KUKA KRL program: EPS_2_25694_RR02_A_20260114065911.src

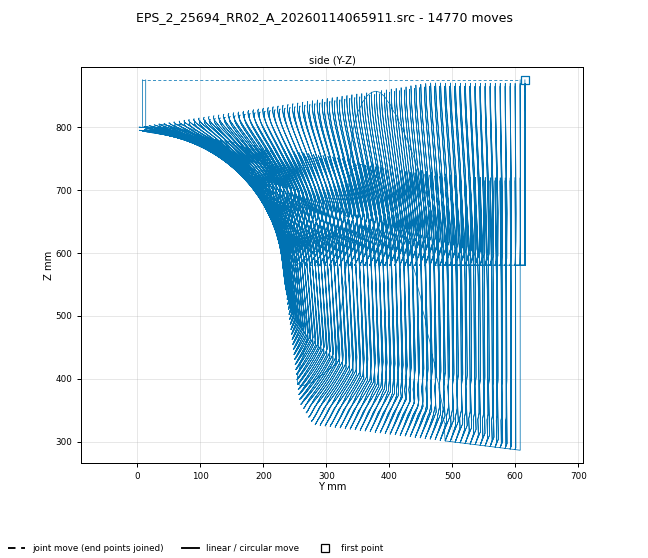
[picture p0: tool path of EPS_2_25694_RR02_A_20260114065911.src, 14770 of 14772 moves have a stored position in this frame; points joined in program order, loops and branches not executed]
&ACCESS RVP
&REL 4
&COMMENT QRS 19112012
&PARAM EDITMASK = *
DEF PART()
EXT BAS (BAS_COMMAND :IN,REAL :IN )
INT I
BAS (#INITMOV,0 )

;KUKA QRS Post kuka4.cps  Date:22-06-2017 !

File_ID=2963

QRS_PRE_INIT()

;Init var - Until changes are made in qrs_pre_init
Outlet_Square_prg=0
Inlet_1_Square_prg=0
Inlet_2_Square_prg=0
Inlet_3_Square_prg=0
Inlet_4_Square_prg=0
Inlet_5_Square_prg=0

Outlet_1={X 0.000, Y 466.000, Z 636.500, B 0.000, E1 0.000 }
Inlet_1={X 0.000, Y 521.440, Z 392.000, B 0.000, E1 180.000 }
Outlet_1_type=457
Inlet_1_type=366
;QRS#1=Sidecore dimensions
;QRS#2=450-18" Concrete
;QRS#3=375-15" PVC SDR 35
;QRS#4=
;QRS#5=
;QRS#6=
;QRS#7=
;QRS#8=
;QRS#9=28A PSX-2
;QRS#10=20Y PSX
;QRS#11=
;QRS#12=
;QRS#13=
;QRS#14=
;QRS#15=
;QRS#16=1220x127x1219 4'
;QRS#17=EPS Height
;QRS#18=865
;QRS#19=*
;QRS#20= UPDATED VERSION 22-06-2017
;QRS#21=*
Outlet_Square=0250
Inlet_1_Square=0250
Inlet_2_Square=0
Inlet_3_Square=0
Inlet_4_Square=0
Inlet_5_Square=0
Mill_Square=1
Outlet_Square_Prg=274
Inlet_1_Square_prg=252

QRS_INIT()

$ADVANCE=5

; T1
PTP {E1 172.637,E2 172.637}
PTP {X 0,Y 615.384,A -85,B 0,C 180,E1 172.637,E2 172.637,E3 0,E4 0,E5 0,E6 0}
QRS_SPEED_INIT()
LIN {X 0,Y 615.384,Z 875,A -85,B 0,C 180,E1 172.637,E2 172.637,E3 0,E4 0,E5 0,E6 0} C_VEL
LIN {X 0,Y 615.384,Z 582.66,A -85,B 0,C 180,E1 172.637,E2 172.637} C_VEL
LIN {X 0,Y 615.412,Z 580.66,A -85,B 0,C 180,E1 172.823,E2 172.823} C_VEL
LIN {X 0,Y 615.825,Z 580.66,A -85,B 0,C 180,E1 174.193,E2 174.193} C_VEL
LIN {X 0,Y 615.841,Z 580.66,A -85,B 0,C 180,E1 178.841,E2 178.841} C_VEL
LIN {X 0,Y 615.793,Z 580.66,A -85,B 0,C 180,E1 183.481,E2 183.481} C_VEL
LIN {X 0,Y 615.82,Z 580.66,A -85,B 0,C 180,E1 188.143,E2 188.143} C_VEL
LIN {X 0,Y 615.802,Z 580.66,A -85,B 0,C 180,E1 192.862,E2 192.862} C_VEL
LIN {X 0,Y 615.751,Z 580.66,A -85,B 0,C 180,E1 197.672,E2 197.672} C_VEL
LIN {X 0,Y 615.756,Z 580.66,A -85,B 0,C 180,E1 197.985,E2 197.985} C_VEL
LIN {X 0,Y 615.766,Z 580.66,A -85,B 0,C 180,E1 202.613,E2 202.613} C_VEL
LIN {X 0,Y 615.233,Z 580.66,A -85,B 0,C 180,E1 205.173,E2 205.173} C_VEL
LIN {X 0,Y 615.723,Z 580.66,A -85,B 0,C 180,E1 207.742,E2 207.742} C_VEL
LIN {X 0,Y 615.16,Z 580.66,A -85,B 0,C 180,E1 210.426,E2 210.426} C_VEL
LIN {X 0,Y 615.691,Z 580.66,A -85,B 0,C 180,E1 213.125,E2 213.125} C_VEL
LIN {X 0,Y 615.621,Z 580.66,A -85,B 0,C 180,E1 213.912,E2 213.912} C_VEL
LIN {X 0,Y 615.656,Z 580.66,A -85,B 0,C 180,E1 218.863,E2 218.863} C_VEL
LIN {X 0,Y 615.25,Z 580.66,A -85,B 0,C 180,E1 221.943,E2 221.943} C_VEL
LIN {X 0,Y 615.658,Z 580.66,A -85,B 0,C 180,E1 224.895,E2 224.895} C_VEL
LIN {X 0,Y 615.649,Z 580.66,A -85,B 0,C 180,E1 228.497,E2 228.497} C_VEL
LIN {X 0,Y 615.377,Z 580.66,A -85,B 0,C 180,E1 231.117,E2 231.117} C_VEL
LIN {X 0,Y 615.425,Z 580.66,A -85,B 0,C 180,E1 232.156,E2 232.156} C_VEL
LIN {X 0,Y 615.687,Z 580.66,A -85,B 0,C 180,E1 234.06,E2 234.06} C_VEL
LIN {X 0,Y 615.153,Z 580.66,A -85,B 0,C 180,E1 236.843,E2 236.843} C_VEL
LIN {X 0,Y 615.758,Z 580.66,A -85,B 0,C 180,E1 239.607,E2 239.607} C_VEL
LIN {X 0,Y 615.721,Z 580.66,A -85,B 0,C 180,E1 243.936,E2 243.936} C_VEL
LIN {X 0,Y 615.733,Z 580.66,A -85,B 0,C 180,E1 244.38,E2 244.38} C_VEL
LIN {X 0,Y 614.989,Z 580.66,A -85,B 0,C 180,E1 244.523,E2 244.523} C_VEL
LIN {X 0,Y 614.799,Z 580.769,A -85,B 0,C 180,E1 244.548,E2 244.548} C_VEL
LIN {X 0,Y 615.5,Z 597.034,A -85,B 0,C 180,E1 244.785,E2 244.785} C_VEL
LIN {X 0,Y 615.746,Z 643.934,A -85,B 0,C 180,E1 245.388,E2 245.388} C_VEL
LIN {X 0,Y 615.746,Z 656.529,A -85,B 0,C 180,E1 245.585,E2 245.585} C_VEL
LIN {X 0,Y 615.551,Z 668.878,A -85,B 0,C 180,E1 245.832,E2 245.832} C_VEL
LIN {X 0,Y 615.688,Z 680.202,A -85,B 0,C 180,E1 246.128,E2 246.128} C_VEL
LIN {X 0,Y 615.662,Z 691.181,A -85,B 0,C 180,E1 246.461,E2 246.461} C_VEL
LIN {X 0,Y 615.686,Z 701.114,A -85,B 0,C 180,E1 246.809,E2 246.809} C_VEL
LIN {X 0,Y 615.746,Z 713.854,A -85,B 0,C 180,E1 247.329,E2 247.329} C_VEL
LIN {X 0,Y 615.681,Z 724.625,A -85,B 0,C 180,E1 247.824,E2 247.824} C_VEL
LIN {X 0,Y 615.745,Z 734.343,A -85,B 0,C 180,E1 248.326,E2 248.326} C_VEL
LIN {X 0,Y 615.763,Z 745.218,A -85,B 0,C 180,E1 248.949,E2 248.949} C_VEL
LIN {X 0,Y 615.754,Z 755.026,A -85,B 0,C 180,E1 249.568,E2 249.568} C_VEL
LIN {X 0,Y 615.75,Z 764.993,A -85,B 0,C 180,E1 250.263,E2 250.263} C_VEL
LIN {X 0,Y 615.755,Z 774.06,A -85,B 0,C 180,E1 250.954,E2 250.954} C_VEL
LIN {X 0,Y 615.778,Z 783.429,A -85,B 0,C 180,E1 251.737,E2 251.737} C_VEL
LIN {X 0,Y 615.741,Z 791.079,A -85,B 0,C 180,E1 252.429,E2 252.429} C_VEL
LIN {X 0,Y 615.699,Z 798.268,A -85,B 0,C 180,E1 253.129,E2 253.129} C_VEL
LIN {X 0,Y 615.745,Z 806.234,A -85,B 0,C 180,E1 253.979,E2 253.979} C_VEL
LIN {X 0,Y 615.811,Z 812.886,A -85,B 0,C 180,E1 254.748,E2 254.748} C_VEL
LIN {X 0,Y 615.686,Z 820.033,A -85,B 0,C 180,E1 255.645,E2 255.645} C_VEL
LIN {X 0,Y 615.678,Z 826.532,A -85,B 0,C 180,E1 256.541,E2 256.541} C_VEL
LIN {X 0,Y 615.8,Z 832.432,A -85,B 0,C 180,E1 257.436,E2 257.436} C_VEL
LIN {X 0,Y 615.696,Z 837.811,A -85,B 0,C 180,E1 258.323,E2 258.323} C_VEL
LIN {X 0,Y 615.617,Z 844.151,A -85,B 0,C 180,E1 259.503,E2 259.503} C_VEL
LIN {X 0,Y 615.751,Z 848.397,A -85,B 0,C 180,E1 260.389,E2 260.389} C_VEL
LIN {X 0,Y 615.781,Z 852.167,A -85,B 0,C 180,E1 261.27,E2 261.27} C_VEL
LIN {X 0,Y 615.632,Z 857.066,A -85,B 0,C 180,E1 262.574,E2 262.574} C_VEL
LIN {X 0,Y 615.761,Z 860.68,A -85,B 0,C 180,E1 263.748,E2 263.748} C_VEL
LIN {X 0,Y 615.831,Z 861.858,A -85,B 0,C 180,E1 264.193,E2 264.193} C_VEL
LIN {X 0,Y 615.724,Z 863.1,A -85,B 0,C 180,E1 264.658,E2 264.658} C_VEL
LIN {X 0,Y 615.59,Z 865.15,A -85,B 0,C 180,E1 265.588,E2 265.588} C_VEL
LIN {X 0,Y 615.604,Z 866.752,A -85,B 0,C 180,E1 266.518,E2 266.518} C_VEL
LIN {X 0,Y 615.789,Z 867.942,A -85,B 0,C 180,E1 267.448,E2 267.448} C_VEL
LIN {X 0,Y 615.603,Z 869.162,A -85,B 0,C 180,E1 268.84,E2 268.84} C_VEL
LIN {X 0,Y 615.628,Z 869.418,A -85,B 0,C 180,E1 270.232,E2 270.232} C_VEL
LIN {X 0,Y 615.832,Z 869.118,A -85,B 0,C 180,E1 271.159,E2 271.159} C_VEL
LIN {X 0,Y 615.718,Z 868.484,A -85,B 0,C 180,E1 272.087,E2 272.087} C_VEL
LIN {X 0,Y 615.795,Z 866.717,A -85,B 0,C 180,E1 273.48,E2 273.48} C_VEL
LIN {X 0,Y 615.708,Z 865.13,A -85,B 0,C 180,E1 274.411,E2 274.411} C_VEL
LIN {X 0,Y 615.577,Z 863.127,A -85,B 0,C 180,E1 275.343,E2 275.343} C_VEL
LIN {X 0,Y 615.645,Z 860.601,A -85,B 0,C 180,E1 276.29,E2 276.29} C_VEL
LIN {X 0,Y 615.806,Z 856.594,A -85,B 0,C 180,E1 277.559,E2 277.559} C_VEL
LIN {X 0,Y 615.635,Z 852.191,A -85,B 0,C 180,E1 278.731,E2 278.731} C_VEL
LIN {X 0,Y 615.664,Z 848.411,A -85,B 0,C 180,E1 279.612,E2 279.612} C_VEL
LIN {X 0,Y 615.797,Z 842.63,A -85,B 0,C 180,E1 280.788,E2 280.788} C_VEL
LIN {X 0,Y 615.635,Z 837.82,A -85,B 0,C 180,E1 281.678,E2 281.678} C_VEL
LIN {X 0,Y 615.632,Z 832.452,A -85,B 0,C 180,E1 282.567,E2 282.567} C_VEL
LIN {X 0,Y 615.823,Z 824.412,A -85,B 0,C 180,E1 283.754,E2 283.754} C_VEL
LIN {X 0,Y 615.734,Z 817.716,A -85,B 0,C 180,E1 284.653,E2 284.653} C_VEL
LIN {X 0,Y 615.702,Z 810.34,A -85,B 0,C 180,E1 285.554,E2 285.554} C_VEL
LIN {X 0,Y 615.782,Z 803.643,A -85,B 0,C 180,E1 286.305,E2 286.305} C_VEL
LIN {X 0,Y 615.769,Z 795.301,A -85,B 0,C 180,E1 287.164,E2 287.164} C_VEL
LIN {X 0,Y 615.716,Z 786.769,A -85,B 0,C 180,E1 287.969,E2 287.969} C_VEL
LIN {X 0,Y 615.738,Z 778.66,A -85,B 0,C 180,E1 288.672,E2 288.672} C_VEL
LIN {X 0,Y 615.745,Z 770.145,A -85,B 0,C 180,E1 289.353,E2 289.353} C_VEL
LIN {X 0,Y 615.75,Z 760.692,A -85,B 0,C 180,E1 290.045,E2 290.045} C_VEL
LIN {X 0,Y 615.742,Z 751.477,A -85,B 0,C 180,E1 290.664,E2 290.664} C_VEL
LIN {X 0,Y 615.715,Z 741.286,A -85,B 0,C 180,E1 291.286,E2 291.286} C_VEL
LIN {X 0,Y 615.749,Z 731.423,A -85,B 0,C 180,E1 291.83,E2 291.83} C_VEL
LIN {X 0,Y 615.746,Z 720.95,A -85,B 0,C 180,E1 292.351,E2 292.351} C_VEL
LIN {X 0,Y 615.698,Z 709.84,A -85,B 0,C 180,E1 292.845,E2 292.845} C_VEL
LIN {X 0,Y 615.669,Z 699.566,A -85,B 0,C 180,E1 293.249,E2 293.249} C_VEL
LIN {X 0,Y 615.734,Z 686.394,A -85,B 0,C 180,E1 293.687,E2 293.687} C_VEL
LIN {X 0,Y 615.669,Z 674.855,A -85,B 0,C 180,E1 294.016,E2 294.016} C_VEL
LIN {X 0,Y 615.62,Z 666.572,A -85,B 0,C 180,E1 294.221,E2 294.221} C_VEL
LIN {X 0,Y 615.767,Z 652.574,A -85,B 0,C 180,E1 294.483,E2 294.483} C_VEL
LIN {X 0,Y 615.685,Z 635.543,A -85,B 0,C 180,E1 294.722,E2 294.722} C_VEL
LIN {X 0,Y 615.162,Z 597.63,A -85,B 0,C 180,E1 295.223,E2 295.223} C_VEL
LIN {X 0,Y 614.785,Z 580.66,A -85,B 0,C 180,E1 295.457,E2 295.457} C_VEL
LIN {X 0,Y 615.85,Z 580.66,A -85,B 0,C 180,E1 295.73,E2 295.73} C_VEL
LIN {X 0,Y 615.813,Z 580.66,A -85,B 0,C 180,E1 297.736,E2 297.736} C_VEL
LIN {X 0,Y 615.182,Z 580.66,A -85,B 0,C 180,E1 300.424,E2 300.424} C_VEL
LIN {X 0,Y 615.704,Z 580.66,A -85,B 0,C 180,E1 303.123,E2 303.123} C_VEL
LIN {X 0,Y 615.639,Z 580.66,A -85,B 0,C 180,E1 303.912,E2 303.912} C_VEL
LIN {X 0,Y 615.658,Z 580.66,A -85,B 0,C 180,E1 308.862,E2 308.862} C_VEL
LIN {X 0,Y 615.25,Z 580.66,A -85,B 0,C 180,E1 311.941,E2 311.941} C_VEL
LIN {X 0,Y 615.666,Z 580.66,A -85,B 0,C 180,E1 314.894,E2 314.894} C_VEL
LIN {X 0,Y 615.661,Z 580.66,A -85,B 0,C 180,E1 318.493,E2 318.493} C_VEL
LIN {X 0,Y 615.374,Z 580.66,A -85,B 0,C 180,E1 321.115,E2 321.115} C_VEL
LIN {X 0,Y 615.423,Z 580.66,A -85,B 0,C 180,E1 322.154,E2 322.154} C_VEL
LIN {X 0,Y 615.672,Z 580.66,A -85,B 0,C 180,E1 324.058,E2 324.058} C_VEL
LIN {X 0,Y 615.143,Z 580.66,A -85,B 0,C 180,E1 326.841,E2 326.841} C_VEL
LIN {X 0,Y 615.743,Z 580.66,A -85,B 0,C 180,E1 329.606,E2 329.606} C_VEL
LIN {X 0,Y 615.21,Z 580.66,A -85,B 0,C 180,E1 332.233,E2 332.233} C_VEL
LIN {X 0,Y 615.726,Z 580.66,A -85,B 0,C 180,E1 334.849,E2 334.849} C_VEL
LIN {X 0,Y 615.762,Z 580.66,A -85,B 0,C 180,E1 339.877,E2 339.877} C_VEL
LIN {X 0,Y 615.795,Z 580.66,A -85,B 0,C 180,E1 343.784,E2 343.784} C_VEL
LIN {X 0,Y 615.809,Z 580.66,A -85,B 0,C 180,E1 349.507,E2 349.507} C_VEL
LIN {X 0,Y 615.792,Z 580.66,A -85,B 0,C 180,E1 354.193,E2 354.193} C_VEL
LIN {X 0,Y 615.815,Z 580.66,A -85,B 0,C 180,E1 358.841,E2 358.841} C_VEL
LIN {X 0,Y 615.862,Z 580.66,A -85,B 0,C 180,E1 363.48,E2 363.48} C_VEL
LIN {X 0,Y 615.786,Z 580.66,A -85,B 0,C 180,E1 368.144,E2 368.144} C_VEL
LIN {X 0,Y 615.765,Z 580.66,A -85,B 0,C 180,E1 372.862,E2 372.862} C_VEL
LIN {X 0,Y 615.802,Z 580.66,A -85,B 0,C 180,E1 377.67,E2 377.67} C_VEL
LIN {X 0,Y 615.801,Z 580.66,A -85,B 0,C 180,E1 377.999,E2 377.999} C_VEL
LIN {X 0,Y 615.737,Z 580.66,A -85,B 0,C 180,E1 382.614,E2 382.614} C_VEL
LIN {X 0,Y 615.212,Z 580.66,A -85,B 0,C 180,E1 385.174,E2 385.174} C_VEL
LIN {X 0,Y 615.723,Z 580.66,A -85,B 0,C 180,E1 387.742,E2 387.742} C_VEL
LIN {X 0,Y 615.169,Z 580.66,A -85,B 0,C 180,E1 390.426,E2 390.426} C_VEL
LIN {X 0,Y 615.697,Z 580.66,A -85,B 0,C 180,E1 393.125,E2 393.125} C_VEL
LIN {X 0,Y 615.637,Z 580.66,A -85,B 0,C 180,E1 393.915,E2 393.915} C_VEL
LIN {X 0,Y 615.621,Z 580.66,A -85,B 0,C 180,E1 398.866,E2 398.866} C_VEL
LIN {X 0,Y 615.224,Z 580.66,A -85,B 0,C 180,E1 401.945,E2 401.945} C_VEL
LIN {X 0,Y 615.653,Z 580.66,A -85,B 0,C 180,E1 404.895,E2 404.895} C_VEL
LIN {X 0,Y 615.628,Z 580.66,A -85,B 0,C 180,E1 408.499,E2 408.499} C_VEL
LIN {X 0,Y 615.36,Z 580.66,A -85,B 0,C 180,E1 411.116,E2 411.116} C_VEL
LIN {X 0,Y 615.418,Z 580.66,A -85,B 0,C 180,E1 412.157,E2 412.157} C_VEL
LIN {X 0,Y 615.69,Z 580.66,A -85,B 0,C 180,E1 414.061,E2 414.061} C_VEL
LIN {X 0,Y 615.128,Z 580.66,A -85,B 0,C 180,E1 416.842,E2 416.842} C_VEL
LIN {X 0,Y 615.699,Z 580.66,A -85,B 0,C 180,E1 419.605,E2 419.605} C_VEL
LIN {X 0,Y 615.208,Z 580.66,A -85,B 0,C 180,E1 422.234,E2 422.234} C_VEL
LIN {X 0,Y 615.756,Z 580.66,A -85,B 0,C 180,E1 424.851,E2 424.851} C_VEL
LIN {X 0,Y 615.821,Z 580.66,A -85,B 0,C 180,E1 429.88,E2 429.88} C_VEL
LIN {X 0,Y 615.638,Z 580.69,A -85,B 0,C 180,E1 431.013,E2 431.013} C_VEL
LIN {X 0,Y 615.768,Z 591.798,A -85,B 0,C 180,E1 431.458,E2 431.458} C_VEL
LIN {X 0,Y 615.772,Z 600.905,A -85,B 0,C 180,E1 431.871,E2 431.871} C_VEL
LIN {X 0,Y 615.729,Z 609.887,A -85,B 0,C 180,E1 432.328,E2 432.328} C_VEL
LIN {X 0,Y 615.771,Z 617.761,A -85,B 0,C 180,E1 432.774,E2 432.774} C_VEL
LIN {X 0,Y 615.774,Z 624.953,A -85,B 0,C 180,E1 433.218,E2 433.218} C_VEL
LIN {X 0,Y 615.803,Z 633.619,A -85,B 0,C 180,E1 433.81,E2 433.81} C_VEL
LIN {X 0,Y 615.788,Z 641.35,A -85,B 0,C 180,E1 434.39,E2 434.39} C_VEL
LIN {X 0,Y 615.765,Z 649.322,A -85,B 0,C 180,E1 435.048,E2 435.048} C_VEL
LIN {X 0,Y 615.775,Z 655.958,A -85,B 0,C 180,E1 435.647,E2 435.647} C_VEL
LIN {X 0,Y 615.829,Z 663.488,A -85,B 0,C 180,E1 436.395,E2 436.395} C_VEL
LIN {X 0,Y 615.772,Z 668.99,A -85,B 0,C 180,E1 436.99,E2 436.99} C_VEL
LIN {X 0,Y 615.717,Z 675.289,A -85,B 0,C 180,E1 437.731,E2 437.731} C_VEL
LIN {X 0,Y 615.762,Z 681.001,A -85,B 0,C 180,E1 438.473,E2 438.473} C_VEL
LIN {X 0,Y 615.83,Z 686.181,A -85,B 0,C 180,E1 439.213,E2 439.213} C_VEL
LIN {X 0,Y 615.701,Z 691.8,A -85,B 0,C 180,E1 440.094,E2 440.094} C_VEL
LIN {X 0,Y 615.678,Z 695.184,A -85,B 0,C 180,E1 440.682,E2 440.682} C_VEL
LIN {X 0,Y 615.763,Z 699.755,A -85,B 0,C 180,E1 441.564,E2 441.564} C_VEL
LIN {X 0,Y 615.828,Z 702.587,A -85,B 0,C 180,E1 442.164,E2 442.164} C_VEL
LIN {X 0,Y 615.7,Z 705.584,A -85,B 0,C 180,E1 442.857,E2 442.857} C_VEL
LIN {X 0,Y 615.634,Z 708.833,A -85,B 0,C 180,E1 443.718,E2 443.718} C_VEL
LIN {X 0,Y 615.72,Z 711.829,A -85,B 0,C 180,E1 444.658,E2 444.658} C_VEL
LIN {X 0,Y 615.799,Z 714.279,A -85,B 0,C 180,E1 445.59,E2 445.59} C_VEL
LIN {X 0,Y 615.646,Z 716.272,A -85,B 0,C 180,E1 446.519,E2 446.519} C_VEL
LIN {X 0,Y 615.657,Z 717.751,A -85,B 0,C 180,E1 447.448,E2 447.448} C_VEL
LIN {X 0,Y 615.718,Z 718.288,A -85,B 0,C 180,E1 447.913,E2 447.913} C_VEL
LIN {X 0,Y 615.776,Z 719.068,A -85,B 0,C 180,E1 448.841,E2 448.841} C_VEL
LIN {X 0,Y 615.635,Z 719.428,A -85,B 0,C 180,E1 449.768,E2 449.768} C_VEL
LIN {X 0,Y 615.625,Z 719.408,A -85,B 0,C 180,E1 450.232,E2 450.232} C_VEL
LIN {X 0,Y 615.726,Z 719.014,A -85,B 0,C 180,E1 451.16,E2 451.16} C_VEL
LIN {X 0,Y 615.709,Z 717.635,A -85,B 0,C 180,E1 452.552,E2 452.552} C_VEL
LIN {X 0,Y 615.64,Z 716.119,A -85,B 0,C 180,E1 453.481,E2 453.481} C_VEL
LIN {X 0,Y 615.741,Z 714.08,A -85,B 0,C 180,E1 454.411,E2 454.411} C_VEL
LIN {X 0,Y 615.791,Z 711.544,A -85,B 0,C 180,E1 455.341,E2 455.341} C_VEL
LIN {X 0,Y 615.685,Z 708.479,A -85,B 0,C 180,E1 456.284,E2 456.284} C_VEL
LIN {X 0,Y 615.769,Z 703.979,A -85,B 0,C 180,E1 457.424,E2 457.424} C_VEL
LIN {X 0,Y 615.81,Z 700.733,A -85,B 0,C 180,E1 458.143,E2 458.143} C_VEL
LIN {X 0,Y 615.718,Z 697.886,A -85,B 0,C 180,E1 458.731,E2 458.731} C_VEL
LIN {X 0,Y 615.682,Z 693.041,A -85,B 0,C 180,E1 459.612,E2 459.612} C_VEL
LIN {X 0,Y 615.79,Z 687.56,A -85,B 0,C 180,E1 460.494,E2 460.494} C_VEL
LIN {X 0,Y 615.811,Z 682.514,A -85,B 0,C 180,E1 461.231,E2 461.231} C_VEL
LIN {X 0,Y 615.725,Z 676.961,A -85,B 0,C 180,E1 461.972,E2 461.972} C_VEL
LIN {X 0,Y 615.74,Z 670.826,A -85,B 0,C 180,E1 462.714,E2 462.714} C_VEL
LIN {X 0,Y 615.83,Z 664.055,A -85,B 0,C 180,E1 463.456,E2 463.456} C_VEL
LIN {X 0,Y 615.807,Z 658.152,A -85,B 0,C 180,E1 464.053,E2 464.053} C_VEL
LIN {X 0,Y 615.764,Z 651.723,A -85,B 0,C 180,E1 464.653,E2 464.653} C_VEL
LIN {X 0,Y 615.786,Z 644.696,A -85,B 0,C 180,E1 465.252,E2 465.252} C_VEL
LIN {X 0,Y 615.794,Z 636.939,A -85,B 0,C 180,E1 465.857,E2 465.857} C_VEL
LIN {X 0,Y 615.802,Z 629.564,A -85,B 0,C 180,E1 466.384,E2 466.384} C_VEL
LIN {X 0,Y 615.782,Z 622.271,A -85,B 0,C 180,E1 466.862,E2 466.862} C_VEL
LIN {X 0,Y 615.747,Z 613.78,A -85,B 0,C 180,E1 467.368,E2 467.368} C_VEL
LIN {X 0,Y 615.782,Z 604.229,A -85,B 0,C 180,E1 467.875,E2 467.875} C_VEL
LIN {X 0,Y 615.762,Z 594.955,A -85,B 0,C 180,E1 468.314,E2 468.314} C_VEL
LIN {X 0,Y 615.677,Z 586.78,A -85,B 0,C 180,E1 468.661,E2 468.661} C_VEL
LIN {X 0,Y 615.567,Z 580.66,A -85,B 0,C 180,E1 468.91,E2 468.91} C_VEL
LIN {X 0,Y 615.866,Z 580.66,A -85,B 0,C 180,E1 469.1,E2 469.1} C_VEL
LIN {X 0,Y 615.851,Z 580.66,A -85,B 0,C 180,E1 470.119,E2 470.119} C_VEL
LIN {X 0,Y 615.763,Z 580.66,A -85,B 0,C 180,E1 475.149,E2 475.149} C_VEL
LIN {X 0,Y 615.383,Z 580.66,A -85,B 0,C 180,E1 479.455,E2 479.455} C_VEL
LIN {X 0,Y 615.701,Z 580.66,A -85,B 0,C 180,E1 480.396,E2 480.396} C_VEL
LIN {X 0,Y 615.131,Z 580.66,A -85,B 0,C 180,E1 483.841,E2 483.841} C_VEL
LIN {X 0,Y 615.679,Z 580.66,A -85,B 0,C 180,E1 485.941,E2 485.941} C_VEL
LIN {X 0,Y 615.645,Z 580.66,A -85,B 0,C 180,E1 487.87,E2 487.87} C_VEL
LIN {X 0,Y 615.733,Z 580.66,A -85,B 0,C 180,E1 488.856,E2 488.856} C_VEL
LIN {X 0,Y 615.227,Z 580.66,A -85,B 0,C 180,E1 491.943,E2 491.943} C_VEL
LIN {X 0,Y 615.643,Z 580.66,A -85,B 0,C 180,E1 494.892,E2 494.892} C_VEL
LIN {X 0,Y 615.619,Z 580.66,A -85,B 0,C 180,E1 498.498,E2 498.498} C_VEL
LIN {X 0,Y 615.352,Z 580.66,A -85,B 0,C 180,E1 501.114,E2 501.114} C_VEL
LIN {X 0,Y 615.402,Z 580.66,A -85,B 0,C 180,E1 502.157,E2 502.157} C_VEL
LIN {X 0,Y 615.677,Z 580.66,A -85,B 0,C 180,E1 504.058,E2 504.058} C_VEL
LIN {X 0,Y 615.116,Z 580.66,A -85,B 0,C 180,E1 506.84,E2 506.84} C_VEL
LIN {X 0,Y 615.688,Z 580.66,A -85,B 0,C 180,E1 509.603,E2 509.603} C_VEL
LIN {X 0,Y 615.191,Z 580.66,A -85,B 0,C 180,E1 512.232,E2 512.232} C_VEL
LIN {X 0,Y 615.73,Z 580.66,A -85,B 0,C 180,E1 514.849,E2 514.849} C_VEL
LIN {X 0,Y 615.767,Z 580.66,A -85,B 0,C 180,E1 519.877,E2 519.877} C_VEL
LIN {X 0,Y 615.703,Z 580.66,A -85,B 0,C 180,E1 523.298,E2 523.298} C_VEL
LIN {X 0,Y 615.368,Z 580.66,A -85,B 0,C 180,E1 524.737,E2 524.737} C_VEL
LIN {X 0,Y 615.764,Z 580.66,A -85,B 0,C 180,E1 529.506,E2 529.506} C_VEL
LIN {X 0,Y 615.412,Z 580.66,A -85,B 0,C 180,E1 532.823,E2 532.823} C_VEL
LIN {X 0,Y 612.993,Z 580.66,A -85,B 0,C 180,E1 534.025,E2 534.025} C_VEL
LIN {X 0,Y 607.572,Z 580.66,A -85,B 0,C 180,E1 535.822,E2 535.822} C_VEL
LIN {X 0,Y 607.462,Z 580.66,A -85,B 0,C 180,E1 536.029,E2 536.029} C_VEL
LIN {X 0,Y 607.577,Z 580.66,A -85,B 0,C 180,E1 540.003,E2 540.003} C_VEL
LIN {X 0,Y 607.637,Z 580.66,A -85,B 0,C 180,E1 544.275,E2 544.275} C_VEL
LIN {X 0,Y 607.765,Z 580.66,A -85,B 0,C 180,E1 548.569,E2 548.569} C_VEL
LIN {X 0,Y 607.891,Z 580.66,A -85,B 0,C 180,E1 552.911,E2 552.911} C_VEL
LIN {X 0,Y 607.583,Z 580.66,A -85,B 0,C 180,E1 558.838,E2 558.838} C_VEL
LIN {X 0,Y 607.578,Z 580.66,A -85,B 0,C 180,E1 563.415,E2 563.415} C_VEL
LIN {X 0,Y 607.667,Z 580.66,A -85,B 0,C 180,E1 568.153,E2 568.153} C_VEL
LIN {X 0,Y 607.798,Z 580.66,A -85,B 0,C 180,E1 573.106,E2 573.106} C_VEL
LIN {X 0,Y 607.506,Z 580.66,A -85,B 0,C 180,E1 579.647,E2 579.647} C_VEL
LIN {X 0,Y 607.513,Z 580.66,A -85,B 0,C 180,E1 585.935,E2 585.935} C_VEL
LIN {X 0,Y 607.445,Z 580.66,A -85,B 0,C 180,E1 590.36,E2 590.36} C_VEL
LIN {X 0,Y 607.42,Z 580.66,A -85,B 0,C 180,E1 595.154,E2 595.154} C_VEL
LIN {X 0,Y 607.622,Z 580.66,A -85,B 0,C 180,E1 600.363,E2 600.363} C_VEL
LIN {X 0,Y 607.839,Z 580.66,A -85,B 0,C 180,E1 604.201,E2 604.201} C_VEL
LIN {X 0,Y 608.382,Z 667.344,A -85,B 0,C 180,E1 605.491,E2 605.491} C_VEL
LIN {X 0,Y 608.354,Z 703.719,A -85,B 0,C 180,E1 606.617,E2 606.617} C_VEL
LIN {X 0,Y 608.282,Z 737.923,A -85,B 0,C 180,E1 608.25,E2 608.25} C_VEL
LIN {X 0,Y 608.145,Z 770.079,A -85,B 0,C 180,E1 610.39,E2 610.39} C_VEL
LIN {X 0,Y 607.967,Z 799.54,A -85,B 0,C 180,E1 613.044,E2 613.044} C_VEL
LIN {X 0,Y 607.857,Z 823.986,A -85,B 0,C 180,E1 615.992,E2 615.992} C_VEL
LIN {X 0,Y 607.781,Z 843.899,A -85,B 0,C 180,E1 619.268,E2 619.268} C_VEL
LIN {X 0,Y 607.771,Z 857.372,A -85,B 0,C 180,E1 622.458,E2 622.458} C_VEL
LIN {X 0,Y 607.711,Z 865.993,A -85,B 0,C 180,E1 625.727,E2 625.727} C_VEL
LIN {X 0,Y 607.74,Z 869.51,A -85,B 0,C 180,E1 628.576,E2 628.576} C_VEL
LIN {X 0,Y 607.908,Z 869.511,A -85,B 0,C 180,E1 631.421,E2 631.421} C_VEL
LIN {X 0,Y 607.732,Z 864.491,A -85,B 0,C 180,E1 634.984,E2 634.984} C_VEL
LIN {X 0,Y 607.841,Z 854.945,A -85,B 0,C 180,E1 638.205,E2 638.205} C_VEL
LIN {X 0,Y 607.836,Z 840.029,A -85,B 0,C 180,E1 641.454,E2 641.454} C_VEL
LIN {X 0,Y 607.954,Z 818.446,A -85,B 0,C 180,E1 644.758,E2 644.758} C_VEL
LIN {X 0,Y 608.054,Z 794.059,A -85,B 0,C 180,E1 647.51,E2 647.51} C_VEL
LIN {X 0,Y 608.187,Z 764.379,A -85,B 0,C 180,E1 650.04,E2 650.04} C_VEL
LIN {X 0,Y 608.315,Z 731.059,A -85,B 0,C 180,E1 652.13,E2 652.13} C_VEL
LIN {X 0,Y 608.414,Z 695.709,A -85,B 0,C 180,E1 653.678,E2 653.678} C_VEL
LIN {X 0,Y 608.506,Z 660.926,A -85,B 0,C 180,E1 654.637,E2 654.637} C_VEL
LIN {X 0,Y 607.896,Z 580.66,A -85,B 0,C 180,E1 655.843,E2 655.843} C_VEL
LIN {X 0,Y 607.342,Z 580.66,A -85,B 0,C 180,E1 661.447,E2 661.447} C_VEL
LIN {X 0,Y 607.381,Z 580.66,A -85,B 0,C 180,E1 664.932,E2 664.932} C_VEL
LIN {X 0,Y 607.379,Z 580.66,A -85,B 0,C 180,E1 670.233,E2 670.233} C_VEL
LIN {X 0,Y 607.498,Z 580.66,A -85,B 0,C 180,E1 676.078,E2 676.078} C_VEL
LIN {X 0,Y 607.445,Z 580.66,A -85,B 0,C 180,E1 680.357,E2 680.357} C_VEL
LIN {X 0,Y 607.412,Z 580.66,A -85,B 0,C 180,E1 685.153,E2 685.153} C_VEL
LIN {X 0,Y 607.586,Z 580.66,A -85,B 0,C 180,E1 690.365,E2 690.365} C_VEL
LIN {X 0,Y 607.762,Z 580.66,A -85,B 0,C 180,E1 695.033,E2 695.033} C_VEL
LIN {X 0,Y 607.561,Z 580.66,A -85,B 0,C 180,E1 701.162,E2 701.162} C_VEL
LIN {X 0,Y 607.245,Z 580.66,A -85,B 0,C 180,E1 705.61,E2 705.61} C_VEL
LIN {X 0,Y 607.731,Z 580.66,A -85,B 0,C 180,E1 709.989,E2 709.989} C_VEL
LIN {X 0,Y 607.866,Z 580.66,A -85,B 0,C 180,E1 714.299,E2 714.299} C_VEL
LIN {X 0,Y 607.548,Z 580.66,A -85,B 0,C 180,E1 719.997,E2 719.997} C_VEL
LIN {X 0,Y 607.66,Z 580.66,A -85,B 0,C 180,E1 724.269,E2 724.269} C_VEL
LIN {X 0,Y 607.738,Z 580.66,A -85,B 0,C 180,E1 728.564,E2 728.564} C_VEL
LIN {X 0,Y 607.84,Z 580.66,A -85,B 0,C 180,E1 732.907,E2 732.907} C_VEL
LIN {X 0,Y 607.599,Z 580.66,A -85,B 0,C 180,E1 738.831,E2 738.831} C_VEL
LIN {X 0,Y 607.548,Z 580.66,A -85,B 0,C 180,E1 743.411,E2 743.411} C_VEL
LIN {X 0,Y 607.658,Z 580.66,A -85,B 0,C 180,E1 748.147,E2 748.147} C_VEL
LIN {X 0,Y 607.792,Z 580.66,A -85,B 0,C 180,E1 753.1,E2 753.1} C_VEL
LIN {X 0,Y 607.451,Z 580.66,A -85,B 0,C 180,E1 759.644,E2 759.644} C_VEL
LIN {X 0,Y 607.517,Z 580.66,A -85,B 0,C 180,E1 765.939,E2 765.939} C_VEL
LIN {X 0,Y 607.406,Z 580.66,A -85,B 0,C 180,E1 770.356,E2 770.356} C_VEL
LIN {X 0,Y 607.416,Z 580.66,A -85,B 0,C 180,E1 775.157,E2 775.157} C_VEL
LIN {X 0,Y 607.52,Z 580.66,A -85,B 0,C 180,E1 780.369,E2 780.369} C_VEL
LIN {X 0,Y 607.79,Z 580.66,A -85,B 0,C 180,E1 785.037,E2 785.037} C_VEL
LIN {X 0,Y 607.766,Z 580.719,A -85,B 0,C 180,E1 790.76,E2 790.76} C_VEL
LIN {X 0,Y 608.152,Z 613.595,A -85,B 0,C 180,E1 792.307,E2 792.307} C_VEL
LIN {X 0,Y 608.064,Z 643.207,A -85,B 0,C 180,E1 794.338,E2 794.338} C_VEL
LIN {X 0,Y 608.004,Z 668.258,A -85,B 0,C 180,E1 796.73,E2 796.73} C_VEL
LIN {X 0,Y 607.961,Z 688.91,A -85,B 0,C 180,E1 799.454,E2 799.454} C_VEL
LIN {X 0,Y 607.905,Z 704.867,A -85,B 0,C 180,E1 802.514,E2 802.514} C_VEL
LIN {X 0,Y 607.897,Z 715.202,A -85,B 0,C 180,E1 805.731,E2 805.731} C_VEL
LIN {X 0,Y 607.874,Z 719.452,A -85,B 0,C 180,E1 808.579,E2 808.579} C_VEL
LIN {X 0,Y 607.827,Z 719.387,A -85,B 0,C 180,E1 811.424,E2 811.424} C_VEL
LIN {X 0,Y 607.85,Z 715.002,A -85,B 0,C 180,E1 814.272,E2 814.272} C_VEL
LIN {X 0,Y 607.902,Z 704.943,A -85,B 0,C 180,E1 817.379,E2 817.379} C_VEL
LIN {X 0,Y 607.929,Z 689.459,A -85,B 0,C 180,E1 820.368,E2 820.368} C_VEL
LIN {X 0,Y 607.967,Z 669.048,A -85,B 0,C 180,E1 823.091,E2 823.091} C_VEL
LIN {X 0,Y 608.072,Z 643.161,A -85,B 0,C 180,E1 825.576,E2 825.576} C_VEL
LIN {X 0,Y 608.161,Z 613.607,A -85,B 0,C 180,E1 827.602,E2 827.602} C_VEL
LIN {X 0,Y 607.974,Z 580.66,A -85,B 0,C 180,E1 829.182,E2 829.182} C_VEL
LIN {X 0,Y 607.799,Z 580.66,A -85,B 0,C 180,E1 834.965,E2 834.965} C_VEL
LIN {X 0,Y 607.575,Z 580.66,A -85,B 0,C 180,E1 839.783,E2 839.783} C_VEL
LIN {X 0,Y 607.709,Z 580.66,A -85,B 0,C 180,E1 846.579,E2 846.579} C_VEL
LIN {X 0,Y 607.313,Z 580.66,A -85,B 0,C 180,E1 851.815,E2 851.815} C_VEL
LIN {X 0,Y 607.466,Z 580.66,A -85,B 0,C 180,E1 856.085,E2 856.085} C_VEL
LIN {X 0,Y 607.398,Z 580.66,A -85,B 0,C 180,E1 860.366,E2 860.366} C_VEL
LIN {X 0,Y 607.398,Z 580.66,A -85,B 0,C 180,E1 865.159,E2 865.159} C_VEL
LIN {X 0,Y 607.519,Z 580.66,A -85,B 0,C 180,E1 870.381,E2 870.381} C_VEL
LIN {X 0,Y 607.75,Z 580.66,A -85,B 0,C 180,E1 875.038,E2 875.038} C_VEL
LIN {X 0,Y 607.617,Z 580.66,A -85,B 0,C 180,E1 881.169,E2 881.169} C_VEL
LIN {X 0,Y 607.197,Z 580.66,A -85,B 0,C 180,E1 885.741,E2 885.741} C_VEL
LIN {X 0,Y 607.695,Z 580.66,A -85,B 0,C 180,E1 889.994,E2 889.994} C_VEL
LIN {X 0,Y 607.878,Z 580.66,A -85,B 0,C 180,E1 894.305,E2 894.305} C_VEL
LIN {X 0,Y 607.462,Z 580.66,A -85,B 0,C 180,E1 896.029,E2 896.029} C_VEL
LIN {X 0,Y 603.66,Z 580.66,A -85,B 0,C 180,E1 897.641,E2 897.641} C_VEL
LIN {X 0,Y 599.763,Z 580.66,A -85,B 0,C 180,E1 899.273,E2 899.273} C_VEL
LIN {X 0,Y 599.719,Z 580.66,A -85,B 0,C 180,E1 904.331,E2 904.331} C_VEL
LIN {X 0,Y 599.822,Z 580.66,A -85,B 0,C 180,E1 908.684,E2 908.684} C_VEL
LIN {X 0,Y 599.91,Z 580.66,A -85,B 0,C 180,E1 913.086,E2 913.086} C_VEL
LIN {X 0,Y 599.63,Z 580.66,A -85,B 0,C 180,E1 919.097,E2 919.097} C_VEL
LIN {X 0,Y 599.587,Z 580.66,A -85,B 0,C 180,E1 923.746,E2 923.746} C_VEL
LIN {X 0,Y 599.654,Z 580.66,A -85,B 0,C 180,E1 928.563,E2 928.563} C_VEL
LIN {X 0,Y 599.663,Z 580.66,A -85,B 0,C 180,E1 933.861,E2 933.861} C_VEL
LIN {X 0,Y 599.616,Z 580.66,A -85,B 0,C 180,E1 938.987,E2 938.987} C_VEL
LIN {X 0,Y 599.529,Z 580.66,A -85,B 0,C 180,E1 945.192,E2 945.192} C_VEL
LIN {X 0,Y 599.538,Z 580.66,A -85,B 0,C 180,E1 951.007,E2 951.007} C_VEL
LIN {X 0,Y 599.572,Z 580.66,A -85,B 0,C 180,E1 954.63,E2 954.63} C_VEL
LIN {X 0,Y 599.661,Z 580.66,A -85,B 0,C 180,E1 959.783,E2 959.783} C_VEL
LIN {X 0,Y 599.899,Z 580.66,A -85,B 0,C 180,E1 963.859,E2 963.859} C_VEL
LIN {X 0,Y 601.303,Z 619.202,A -85,B 0,C 180,E1 964.434,E2 964.434} C_VEL
LIN {X 0,Y 601.135,Z 669.7,A -85,B 0,C 180,E1 965.235,E2 965.235} C_VEL
LIN {X 0,Y 601.058,Z 706.112,A -85,B 0,C 180,E1 966.414,E2 966.414} C_VEL
LIN {X 0,Y 600.805,Z 740.395,A -85,B 0,C 180,E1 968.107,E2 968.107} C_VEL
LIN {X 0,Y 600.54,Z 773.011,A -85,B 0,C 180,E1 970.364,E2 970.364} C_VEL
LIN {X 0,Y 600.229,Z 802.039,A -85,B 0,C 180,E1 973.087,E2 973.087} C_VEL
LIN {X 0,Y 600.059,Z 826.589,A -85,B 0,C 180,E1 976.178,E2 976.178} C_VEL
LIN {X 0,Y 599.919,Z 844.856,A -85,B 0,C 180,E1 979.327,E2 979.327} C_VEL
LIN {X 0,Y 599.881,Z 857.537,A -85,B 0,C 180,E1 982.41,E2 982.41} C_VEL
LIN {X 0,Y 599.827,Z 865.992,A -85,B 0,C 180,E1 985.671,E2 985.671} C_VEL
LIN {X 0,Y 599.84,Z 869.51,A -85,B 0,C 180,E1 988.557,E2 988.557} C_VEL
LIN {X 0,Y 600.005,Z 869.512,A -85,B 0,C 180,E1 991.44,E2 991.44} C_VEL
LIN {X 0,Y 599.953,Z 865.997,A -85,B 0,C 180,E1 994.326,E2 994.326} C_VEL
LIN {X 0,Y 599.995,Z 856.28,A -85,B 0,C 180,E1 997.949,E2 997.949} C_VEL
LIN {X 0,Y 600.006,Z 841.936,A -85,B 0,C 180,E1 1001.247,E2 1001.247} C_VEL
LIN {X 0,Y 600.152,Z 822.673,A -85,B 0,C 180,E1 1004.374,E2 1004.374} C_VEL
LIN {X 0,Y 600.36,Z 797.143,A -85,B 0,C 180,E1 1007.435,E2 1007.435} C_VEL
LIN {X 0,Y 600.58,Z 767.761,A -85,B 0,C 180,E1 1010.045,E2 1010.045} C_VEL
LIN {X 0,Y 600.853,Z 734.821,A -85,B 0,C 180,E1 1012.213,E2 1012.213} C_VEL
LIN {X 0,Y 601.098,Z 698.766,A -85,B 0,C 180,E1 1013.876,E2 1013.876} C_VEL
LIN {X 0,Y 601.294,Z 662.551,A -85,B 0,C 180,E1 1014.92,E2 1014.92} C_VEL
LIN {X 0,Y 600.019,Z 580.66,A -85,B 0,C 180,E1 1016.157,E2 1016.157} C_VEL
LIN {X 0,Y 599.517,Z 580.66,A -85,B 0,C 180,E1 1021.906,E2 1021.906} C_VEL
LIN {X 0,Y 599.297,Z 580.66,A -85,B 0,C 180,E1 1026.321,E2 1026.321} C_VEL
LIN {X 0,Y 599.414,Z 580.66,A -85,B 0,C 180,E1 1030.956,E2 1030.956} C_VEL
LIN {X 0,Y 599.572,Z 580.66,A -85,B 0,C 180,E1 1036.87,E2 1036.87} C_VEL
LIN {X 0,Y 599.654,Z 580.66,A -85,B 0,C 180,E1 1042.847,E2 1042.847} C_VEL
LIN {X 0,Y 599.561,Z 580.66,A -85,B 0,C 180,E1 1048.832,E2 1048.832} C_VEL
LIN {X 0,Y 599.828,Z 580.66,A -85,B 0,C 180,E1 1054.902,E2 1054.902} C_VEL
LIN {X 0,Y 599.712,Z 580.66,A -85,B 0,C 180,E1 1060.906,E2 1060.906} C_VEL
LIN {X 0,Y 599.384,Z 580.66,A -85,B 0,C 180,E1 1065.417,E2 1065.417} C_VEL
LIN {X 0,Y 599.79,Z 580.66,A -85,B 0,C 180,E1 1069.855,E2 1069.855} C_VEL
LIN {X 0,Y 599.963,Z 580.66,A -85,B 0,C 180,E1 1074.224,E2 1074.224} C_VEL
LIN {X 0,Y 599.648,Z 580.66,A -85,B 0,C 180,E1 1079.997,E2 1079.997} C_VEL
LIN {X 0,Y 599.758,Z 580.66,A -85,B 0,C 180,E1 1084.326,E2 1084.326} C_VEL
LIN {X 0,Y 599.795,Z 580.66,A -85,B 0,C 180,E1 1088.679,E2 1088.679} C_VEL
LIN {X 0,Y 599.864,Z 580.66,A -85,B 0,C 180,E1 1093.081,E2 1093.081} C_VEL
LIN {X 0,Y 599.649,Z 580.66,A -85,B 0,C 180,E1 1099.091,E2 1099.091} C_VEL
LIN {X 0,Y 599.562,Z 580.66,A -85,B 0,C 180,E1 1103.741,E2 1103.741} C_VEL
LIN {X 0,Y 599.64,Z 580.66,A -85,B 0,C 180,E1 1108.558,E2 1108.558} C_VEL
LIN {X 0,Y 599.66,Z 580.66,A -85,B 0,C 180,E1 1113.865,E2 1113.865} C_VEL
LIN {X 0,Y 599.571,Z 580.66,A -85,B 0,C 180,E1 1118.983,E2 1118.983} C_VEL
LIN {X 0,Y 599.521,Z 580.66,A -85,B 0,C 180,E1 1125.195,E2 1125.195} C_VEL
LIN {X 0,Y 599.528,Z 580.66,A -85,B 0,C 180,E1 1131.01,E2 1131.01} C_VEL
LIN {X 0,Y 599.549,Z 580.66,A -85,B 0,C 180,E1 1134.632,E2 1134.632} C_VEL
LIN {X 0,Y 599.584,Z 580.66,A -85,B 0,C 180,E1 1139.781,E2 1139.781} C_VEL
LIN {X 0,Y 599.843,Z 580.66,A -85,B 0,C 180,E1 1144.892,E2 1144.892} C_VEL
LIN {X 0,Y 599.905,Z 581.167,A -85,B 0,C 180,E1 1150.516,E2 1150.516} C_VEL
LIN {X 0,Y 600.552,Z 611.909,A -85,B 0,C 180,E1 1151.981,E2 1151.981} C_VEL
LIN {X 0,Y 600.407,Z 641.02,A -85,B 0,C 180,E1 1153.953,E2 1153.953} C_VEL
LIN {X 0,Y 600.259,Z 666.652,A -85,B 0,C 180,E1 1156.37,E2 1156.37} C_VEL
LIN {X 0,Y 600.111,Z 688.543,A -85,B 0,C 180,E1 1159.259,E2 1159.259} C_VEL
LIN {X 0,Y 600.067,Z 703.335,A -85,B 0,C 180,E1 1162.052,E2 1162.052} C_VEL
LIN {X 0,Y 599.969,Z 713.421,A -85,B 0,C 180,E1 1164.951,E2 1164.951} C_VEL
LIN {X 0,Y 599.892,Z 717.9,A -85,B 0,C 180,E1 1167.118,E2 1167.118} C_VEL
LIN {X 0,Y 599.855,Z 719.996,A -85,B 0,C 180,E1 1170.001,E2 1170.001} C_VEL
LIN {X 0,Y 599.921,Z 717.748,A -85,B 0,C 180,E1 1172.885,E2 1172.885} C_VEL
LIN {X 0,Y 599.966,Z 709.658,A -85,B 0,C 180,E1 1176.226,E2 1176.226} C_VEL
LIN {X 0,Y 599.963,Z 697.723,A -85,B 0,C 180,E1 1179.045,E2 1179.045} C_VEL
LIN {X 0,Y 600.079,Z 679.46,A -85,B 0,C 180,E1 1181.974,E2 1181.974} C_VEL
LIN {X 0,Y 600.257,Z 655.669,A -85,B 0,C 180,E1 1184.671,E2 1184.671} C_VEL
LIN {X 0,Y 600.485,Z 628.374,A -85,B 0,C 180,E1 1186.897,E2 1186.897} C_VEL
LIN {X 0,Y 600.687,Z 597.419,A -85,B 0,C 180,E1 1188.681,E2 1188.681} C_VEL
LIN {X 0,Y 600.059,Z 580.66,A -85,B 0,C 180,E1 1189.433,E2 1189.433} C_VEL
LIN {X 0,Y 599.764,Z 580.66,A -85,B 0,C 180,E1 1195.323,E2 1195.323} C_VEL
LIN {X 0,Y 599.511,Z 580.66,A -85,B 0,C 180,E1 1201.166,E2 1201.166} C_VEL
LIN {X 0,Y 599.786,Z 580.66,A -85,B 0,C 180,E1 1207.143,E2 1207.143} C_VEL
LIN {X 0,Y 599.418,Z 580.66,A -85,B 0,C 180,E1 1213.118,E2 1213.118} C_VEL
LIN {X 0,Y 599.567,Z 580.66,A -85,B 0,C 180,E1 1219.027,E2 1219.027} C_VEL
LIN {X 0,Y 599.544,Z 580.66,A -85,B 0,C 180,E1 1224.635,E2 1224.635} C_VEL
LIN {X 0,Y 599.578,Z 580.66,A -85,B 0,C 180,E1 1229.784,E2 1229.784} C_VEL
LIN {X 0,Y 599.827,Z 580.66,A -85,B 0,C 180,E1 1234.908,E2 1234.908} C_VEL
LIN {X 0,Y 599.747,Z 580.66,A -85,B 0,C 180,E1 1240.913,E2 1240.913} C_VEL
LIN {X 0,Y 599.363,Z 580.66,A -85,B 0,C 180,E1 1245.422,E2 1245.422} C_VEL
LIN {X 0,Y 599.754,Z 580.66,A -85,B 0,C 180,E1 1249.86,E2 1249.86} C_VEL
LIN {X 0,Y 599.98,Z 580.66,A -85,B 0,C 180,E1 1254.229,E2 1254.229} C_VEL
LIN {X 0,Y 599.763,Z 580.66,A -85,B 0,C 180,E1 1259.273,E2 1259.273} C_VEL
LIN {X 0,Y 595.598,Z 580.66,A -85,B 0,C 180,E1 1260.905,E2 1260.905} C_VEL
LIN {X 0,Y 591.777,Z 580.66,A -85,B 0,C 180,E1 1262.558,E2 1262.558} C_VEL
LIN {X 0,Y 591.882,Z 580.66,A -85,B 0,C 180,E1 1268.801,E2 1268.801} C_VEL
LIN {X 0,Y 591.664,Z 580.66,A -85,B 0,C 180,E1 1274.273,E2 1274.273} C_VEL
LIN {X 0,Y 591.686,Z 580.66,A -85,B 0,C 180,E1 1279.364,E2 1279.364} C_VEL
LIN {X 0,Y 591.618,Z 580.66,A -85,B 0,C 180,E1 1284.086,E2 1284.086} C_VEL
LIN {X 0,Y 591.628,Z 580.66,A -85,B 0,C 180,E1 1288.987,E2 1288.987} C_VEL
LIN {X 0,Y 591.712,Z 580.66,A -85,B 0,C 180,E1 1294.128,E2 1294.128} C_VEL
LIN {X 0,Y 591.532,Z 580.66,A -85,B 0,C 180,E1 1300.068,E2 1300.068} C_VEL
LIN {X 0,Y 591.593,Z 580.66,A -85,B 0,C 180,E1 1305.577,E2 1305.577} C_VEL
LIN {X 0,Y 591.586,Z 580.66,A -85,B 0,C 180,E1 1310.381,E2 1310.381} C_VEL
LIN {X 0,Y 591.495,Z 580.66,A -85,B 0,C 180,E1 1315.858,E2 1315.858} C_VEL
LIN {X 0,Y 591.62,Z 580.66,A -85,B 0,C 180,E1 1321.013,E2 1321.013} C_VEL
LIN {X 0,Y 591.85,Z 580.66,A -85,B 0,C 180,E1 1323.465,E2 1323.465} C_VEL
LIN {X 0,Y 593.747,Z 589.059,A -85,B 0,C 180,E1 1323.687,E2 1323.687} C_VEL
LIN {X 0,Y 594.09,Z 665.062,A -85,B 0,C 180,E1 1324.808,E2 1324.808} C_VEL
LIN {X 0,Y 593.792,Z 702.597,A -85,B 0,C 180,E1 1325.962,E2 1325.962} C_VEL
LIN {X 0,Y 593.425,Z 736.249,A -85,B 0,C 180,E1 1327.578,E2 1327.578} C_VEL
LIN {X 0,Y 592.984,Z 768.313,A -85,B 0,C 180,E1 1329.73,E2 1329.73} C_VEL
LIN {X 0,Y 592.611,Z 797.708,A -85,B 0,C 180,E1 1332.39,E2 1332.39} C_VEL
LIN {X 0,Y 592.298,Z 823.063,A -85,B 0,C 180,E1 1335.486,E2 1335.486} C_VEL
LIN {X 0,Y 592.064,Z 842.953,A -85,B 0,C 180,E1 1338.794,E2 1338.794} C_VEL
LIN {X 0,Y 591.998,Z 857.537,A -85,B 0,C 180,E1 1342.309,E2 1342.309} C_VEL
LIN {X 0,Y 591.931,Z 865.992,A -85,B 0,C 180,E1 1345.613,E2 1345.613} C_VEL
LIN {X 0,Y 591.94,Z 869.51,A -85,B 0,C 180,E1 1348.538,E2 1348.538} C_VEL
LIN {X 0,Y 592.102,Z 869.512,A -85,B 0,C 180,E1 1351.459,E2 1351.459} C_VEL
LIN {X 0,Y 592.04,Z 865.996,A -85,B 0,C 180,E1 1354.384,E2 1354.384} C_VEL
LIN {X 0,Y 592.105,Z 856.28,A -85,B 0,C 180,E1 1358.056,E2 1358.056} C_VEL
LIN {X 0,Y 592.14,Z 841.937,A -85,B 0,C 180,E1 1361.398,E2 1361.398} C_VEL
LIN {X 0,Y 592.337,Z 822.953,A -85,B 0,C 180,E1 1364.529,E2 1364.529} C_VEL
LIN {X 0,Y 592.637,Z 797.585,A -85,B 0,C 180,E1 1367.623,E2 1367.623} C_VEL
LIN {X 0,Y 593.026,Z 768.351,A -85,B 0,C 180,E1 1370.266,E2 1370.266} C_VEL
LIN {X 0,Y 593.411,Z 736.295,A -85,B 0,C 180,E1 1372.42,E2 1372.42} C_VEL
LIN {X 0,Y 593.813,Z 700.458,A -85,B 0,C 180,E1 1374.125,E2 1374.125} C_VEL
LIN {X 0,Y 594.124,Z 663.999,A -85,B 0,C 180,E1 1375.212,E2 1375.212} C_VEL
LIN {X 0,Y 592.931,Z 584.137,A -85,B 0,C 180,E1 1376.418,E2 1376.418} C_VEL
LIN {X 0,Y 592.068,Z 580.66,A -85,B 0,C 180,E1 1376.565,E2 1376.565} C_VEL
LIN {X 0,Y 591.677,Z 580.66,A -85,B 0,C 180,E1 1382.691,E2 1382.691} C_VEL
LIN {X 0,Y 591.527,Z 580.66,A -85,B 0,C 180,E1 1387.748,E2 1387.748} C_VEL
LIN {X 0,Y 591.519,Z 580.66,A -85,B 0,C 180,E1 1393.529,E2 1393.529} C_VEL
LIN {X 0,Y 591.643,Z 580.66,A -85,B 0,C 180,E1 1398.462,E2 1398.462} C_VEL
LIN {X 0,Y 591.709,Z 580.66,A -85,B 0,C 180,E1 1404.088,E2 1404.088} C_VEL
LIN {X 0,Y 591.65,Z 580.66,A -85,B 0,C 180,E1 1410.123,E2 1410.123} C_VEL
LIN {X 0,Y 591.635,Z 580.66,A -85,B 0,C 180,E1 1415.915,E2 1415.915} C_VEL
LIN {X 0,Y 591.802,Z 580.66,A -85,B 0,C 180,E1 1420.64,E2 1420.64} C_VEL
LIN {X 0,Y 591.515,Z 580.66,A -85,B 0,C 180,E1 1425.219,E2 1425.219} C_VEL
LIN {X 0,Y 591.859,Z 580.66,A -85,B 0,C 180,E1 1429.717,E2 1429.717} C_VEL
LIN {X 0,Y 592.027,Z 580.66,A -85,B 0,C 180,E1 1434.146,E2 1434.146} C_VEL
LIN {X 0,Y 591.748,Z 580.66,A -85,B 0,C 180,E1 1439.997,E2 1439.997} C_VEL
LIN {X 0,Y 591.842,Z 580.66,A -85,B 0,C 180,E1 1444.384,E2 1444.384} C_VEL
LIN {X 0,Y 591.854,Z 580.66,A -85,B 0,C 180,E1 1448.796,E2 1448.796} C_VEL
LIN {X 0,Y 591.633,Z 580.66,A -85,B 0,C 180,E1 1454.271,E2 1454.271} C_VEL
LIN {X 0,Y 591.696,Z 580.66,A -85,B 0,C 180,E1 1459.357,E2 1459.357} C_VEL
LIN {X 0,Y 591.601,Z 580.66,A -85,B 0,C 180,E1 1464.081,E2 1464.081} C_VEL
LIN {X 0,Y 591.619,Z 580.66,A -85,B 0,C 180,E1 1468.981,E2 1468.981} C_VEL
LIN {X 0,Y 591.71,Z 580.66,A -85,B 0,C 180,E1 1474.122,E2 1474.122} C_VEL
LIN {X 0,Y 591.494,Z 580.66,A -85,B 0,C 180,E1 1480.068,E2 1480.068} C_VEL
LIN {X 0,Y 591.585,Z 580.66,A -85,B 0,C 180,E1 1485.57,E2 1485.57} C_VEL
LIN {X 0,Y 591.571,Z 580.66,A -85,B 0,C 180,E1 1490.383,E2 1490.383} C_VEL
LIN {X 0,Y 591.474,Z 580.66,A -85,B 0,C 180,E1 1495.86,E2 1495.86} C_VEL
LIN {X 0,Y 591.537,Z 580.66,A -85,B 0,C 180,E1 1501.011,E2 1501.011} C_VEL
LIN {X 0,Y 591.654,Z 580.66,A -85,B 0,C 180,E1 1505.919,E2 1505.919} C_VEL
LIN {X 0,Y 591.971,Z 580.971,A -85,B 0,C 180,E1 1510.237,E2 1510.237} C_VEL
LIN {X 0,Y 593.176,Z 597.36,A -85,B 0,C 180,E1 1510.98,E2 1510.98} C_VEL
LIN {X 0,Y 592.816,Z 628.344,A -85,B 0,C 180,E1 1512.784,E2 1512.784} C_VEL
LIN {X 0,Y 592.532,Z 655.839,A -85,B 0,C 180,E1 1515.059,E2 1515.059} C_VEL
LIN {X 0,Y 592.256,Z 678.794,A -85,B 0,C 180,E1 1517.681,E2 1517.681} C_VEL
LIN {X 0,Y 592.123,Z 696.265,A -85,B 0,C 180,E1 1520.467,E2 1520.467} C_VEL
LIN {X 0,Y 592.011,Z 708.622,A -85,B 0,C 180,E1 1523.303,E2 1523.303} C_VEL
LIN {X 0,Y 592.046,Z 716.71,A -85,B 0,C 180,E1 1526.348,E2 1526.348} C_VEL
LIN {X 0,Y 592.066,Z 719.452,A -85,B 0,C 180,E1 1528.541,E2 1528.541} C_VEL
LIN {X 0,Y 592.022,Z 719.388,A -85,B 0,C 180,E1 1531.462,E2 1531.462} C_VEL
LIN {X 0,Y 592.075,Z 715.005,A -85,B 0,C 180,E1 1534.386,E2 1534.386} C_VEL
LIN {X 0,Y 592.17,Z 704.479,A -85,B 0,C 180,E1 1537.689,E2 1537.689} C_VEL
LIN {X 0,Y 592.267,Z 688.466,A -85,B 0,C 180,E1 1540.806,E2 1540.806} C_VEL
LIN {X 0,Y 592.463,Z 667.782,A -85,B 0,C 180,E1 1543.59,E2 1543.59} C_VEL
LIN {X 0,Y 592.683,Z 642.179,A -85,B 0,C 180,E1 1546.075,E2 1546.075} C_VEL
LIN {X 0,Y 592.992,Z 611.959,A -85,B 0,C 180,E1 1548.164,E2 1548.164} C_VEL
LIN {X 0,Y 592.491,Z 582.999,A -85,B 0,C 180,E1 1549.574,E2 1549.574} C_VEL
LIN {X 0,Y 592.098,Z 580.66,A -85,B 0,C 180,E1 1549.781,E2 1549.781} C_VEL
LIN {X 0,Y 591.743,Z 580.66,A -85,B 0,C 180,E1 1555.691,E2 1555.691} C_VEL
LIN {X 0,Y 591.63,Z 580.66,A -85,B 0,C 180,E1 1560.671,E2 1560.671} C_VEL
LIN {X 0,Y 591.749,Z 580.66,A -85,B 0,C 180,E1 1565.909,E2 1565.909} C_VEL
LIN {X 0,Y 591.574,Z 580.66,A -85,B 0,C 180,E1 1570.082,E2 1570.082} C_VEL
LIN {X 0,Y 591.567,Z 580.66,A -85,B 0,C 180,E1 1575.579,E2 1575.579} C_VEL
LIN {X 0,Y 591.551,Z 580.66,A -85,B 0,C 180,E1 1580.385,E2 1580.385} C_VEL
LIN {X 0,Y 591.627,Z 580.66,A -85,B 0,C 180,E1 1584.703,E2 1584.703} C_VEL
LIN {X 0,Y 591.528,Z 580.66,A -85,B 0,C 180,E1 1591.014,E2 1591.014} C_VEL
LIN {X 0,Y 591.631,Z 580.66,A -85,B 0,C 180,E1 1595.92,E2 1595.92} C_VEL
LIN {X 0,Y 591.83,Z 580.66,A -85,B 0,C 180,E1 1600.647,E2 1600.647} C_VEL
LIN {X 0,Y 591.415,Z 580.66,A -85,B 0,C 180,E1 1605.822,E2 1605.822} C_VEL
LIN {X 0,Y 591.63,Z 580.66,A -85,B 0,C 180,E1 1611.201,E2 1611.201} C_VEL
LIN {X 0,Y 591.713,Z 580.66,A -85,B 0,C 180,E1 1615.615,E2 1615.615} C_VEL
LIN {X 0,Y 591.775,Z 580.66,A -85,B 0,C 180,E1 1620.003,E2 1620.003} C_VEL
LIN {X 0,Y 591.777,Z 580.66,A -85,B 0,C 180,E1 1622.558,E2 1622.558} C_VEL
LIN {X 0,Y 589.335,Z 580.66,A -85,B 0,C 180,E1 1623.807,E2 1623.807} C_VEL
LIN {X 0,Y 583.836,Z 580.66,A -85,B 0,C 180,E1 1625.676,E2 1625.676} C_VEL
LIN {X 0,Y 583.743,Z 580.66,A -85,B 0,C 180,E1 1625.892,E2 1625.892} C_VEL
LIN {X 0,Y 583.738,Z 580.66,A -85,B 0,C 180,E1 1630.799,E2 1630.799} C_VEL
LIN {X 0,Y 583.679,Z 580.66,A -85,B 0,C 180,E1 1634.984,E2 1634.984} C_VEL
LIN {X 0,Y 583.746,Z 580.66,A -85,B 0,C 180,E1 1639.638,E2 1639.638} C_VEL
LIN {X 0,Y 583.66,Z 580.66,A -85,B 0,C 180,E1 1644.436,E2 1644.436} C_VEL
LIN {X 0,Y 583.636,Z 580.66,A -85,B 0,C 180,E1 1649.423,E2 1649.423} C_VEL
LIN {X 0,Y 583.716,Z 580.66,A -85,B 0,C 180,E1 1654.662,E2 1654.662} C_VEL
LIN {X 0,Y 583.598,Z 580.66,A -85,B 0,C 180,E1 1660.271,E2 1660.271} C_VEL
LIN {X 0,Y 583.724,Z 580.66,A -85,B 0,C 180,E1 1666.37,E2 1666.37} C_VEL
LIN {X 0,Y 583.709,Z 580.66,A -85,B 0,C 180,E1 1671.652,E2 1671.652} C_VEL
LIN {X 0,Y 583.578,Z 580.66,A -85,B 0,C 180,E1 1677.112,E2 1677.112} C_VEL
LIN {X 0,Y 583.881,Z 580.66,A -85,B 0,C 180,E1 1683.09,E2 1683.09} C_VEL
LIN {X 0,Y 586.725,Z 591.573,A -85,B 0,C 180,E1 1683.381,E2 1683.381} C_VEL
LIN {X 0,Y 586.901,Z 666.795,A -85,B 0,C 180,E1 1684.517,E2 1684.517} C_VEL
LIN {X 0,Y 586.508,Z 703.723,A -85,B 0,C 180,E1 1685.691,E2 1685.691} C_VEL
LIN {X 0,Y 585.986,Z 738.226,A -85,B 0,C 180,E1 1687.395,E2 1687.395} C_VEL
LIN {X 0,Y 585.409,Z 770.592,A -85,B 0,C 180,E1 1689.636,E2 1689.636} C_VEL
LIN {X 0,Y 584.854,Z 800.04,A -85,B 0,C 180,E1 1692.407,E2 1692.407} C_VEL
LIN {X 0,Y 584.499,Z 824.052,A -85,B 0,C 180,E1 1695.43,E2 1695.43} C_VEL
LIN {X 0,Y 584.244,Z 842.713,A -85,B 0,C 180,E1 1698.595,E2 1698.595} C_VEL
LIN {X 0,Y 584.144,Z 857.536,A -85,B 0,C 180,E1 1702.205,E2 1702.205} C_VEL
LIN {X 0,Y 584.046,Z 865.991,A -85,B 0,C 180,E1 1705.553,E2 1705.553} C_VEL
LIN {X 0,Y 584.063,Z 869.51,A -85,B 0,C 180,E1 1708.518,E2 1708.518} C_VEL
LIN {X 0,Y 584.213,Z 869.512,A -85,B 0,C 180,E1 1711.479,E2 1711.479} C_VEL
LIN {X 0,Y 584.135,Z 865.996,A -85,B 0,C 180,E1 1714.443,E2 1714.443} C_VEL
LIN {X 0,Y 584.23,Z 856.28,A -85,B 0,C 180,E1 1718.165,E2 1718.165} C_VEL
LIN {X 0,Y 584.268,Z 841.29,A -85,B 0,C 180,E1 1721.679,E2 1721.679} C_VEL
LIN {X 0,Y 584.529,Z 821.343,A -85,B 0,C 180,E1 1724.959,E2 1724.959} C_VEL
LIN {X 0,Y 584.949,Z 795.967,A -85,B 0,C 180,E1 1728.031,E2 1728.031} C_VEL
LIN {X 0,Y 585.494,Z 766.886,A -85,B 0,C 180,E1 1730.654,E2 1730.654} C_VEL
LIN {X 0,Y 586.08,Z 733.781,A -85,B 0,C 180,E1 1732.865,E2 1732.865} C_VEL
LIN {X 0,Y 586.564,Z 698.771,A -85,B 0,C 180,E1 1734.506,E2 1734.506} C_VEL
LIN {X 0,Y 586.998,Z 662.622,A -85,B 0,C 180,E1 1735.569,E2 1735.569} C_VEL
LIN {X 0,Y 585.943,Z 586.474,A -85,B 0,C 180,E1 1736.726,E2 1736.726} C_VEL
LIN {X 0,Y 584.141,Z 580.66,A -85,B 0,C 180,E1 1736.923,E2 1736.923} C_VEL
LIN {X 0,Y 583.82,Z 580.66,A -85,B 0,C 180,E1 1744.201,E2 1744.201} C_VEL
LIN {X 0,Y 583.6,Z 580.66,A -85,B 0,C 180,E1 1750.268,E2 1750.268} C_VEL
LIN {X 0,Y 583.752,Z 580.66,A -85,B 0,C 180,E1 1756.364,E2 1756.364} C_VEL
LIN {X 0,Y 583.706,Z 580.66,A -85,B 0,C 180,E1 1761.652,E2 1761.652} C_VEL
LIN {X 0,Y 583.571,Z 580.66,A -85,B 0,C 180,E1 1767.111,E2 1767.111} C_VEL
LIN {X 0,Y 583.621,Z 580.66,A -85,B 0,C 180,E1 1772.263,E2 1772.263} C_VEL
LIN {X 0,Y 583.587,Z 580.66,A -85,B 0,C 180,E1 1777.178,E2 1777.178} C_VEL
LIN {X 0,Y 583.858,Z 580.66,A -85,B 0,C 180,E1 1781.931,E2 1781.931} C_VEL
LIN {X 0,Y 583.674,Z 580.66,A -85,B 0,C 180,E1 1788.062,E2 1788.062} C_VEL
LIN {X 0,Y 584.108,Z 580.66,A -85,B 0,C 180,E1 1794.066,E2 1794.066} C_VEL
LIN {X 0,Y 583.869,Z 580.66,A -85,B 0,C 180,E1 1799.997,E2 1799.997} C_VEL
LIN {X 0,Y 583.939,Z 580.66,A -85,B 0,C 180,E1 1804.443,E2 1804.443} C_VEL
LIN {X 0,Y 583.918,Z 580.66,A -85,B 0,C 180,E1 1808.916,E2 1808.916} C_VEL
LIN {X 0,Y 583.953,Z 580.66,A -85,B 0,C 180,E1 1813.444,E2 1813.444} C_VEL
LIN {X 0,Y 583.922,Z 580.66,A -85,B 0,C 180,E1 1818.061,E2 1818.061} C_VEL
LIN {X 0,Y 583.791,Z 580.66,A -85,B 0,C 180,E1 1822.808,E2 1822.808} C_VEL
LIN {X 0,Y 583.691,Z 580.66,A -85,B 0,C 180,E1 1828.488,E2 1828.488} C_VEL
LIN {X 0,Y 583.705,Z 580.66,A -85,B 0,C 180,E1 1834.656,E2 1834.656} C_VEL
LIN {X 0,Y 583.563,Z 580.66,A -85,B 0,C 180,E1 1840.267,E2 1840.267} C_VEL
LIN {X 0,Y 583.732,Z 580.66,A -85,B 0,C 180,E1 1846.362,E2 1846.362} C_VEL
LIN {X 0,Y 583.694,Z 580.66,A -85,B 0,C 180,E1 1851.654,E2 1851.654} C_VEL
LIN {X 0,Y 583.548,Z 580.66,A -85,B 0,C 180,E1 1857.113,E2 1857.113} C_VEL
LIN {X 0,Y 583.607,Z 580.66,A -85,B 0,C 180,E1 1862.266,E2 1862.266} C_VEL
LIN {X 0,Y 583.616,Z 580.66,A -85,B 0,C 180,E1 1867.182,E2 1867.182} C_VEL
LIN {X 0,Y 584.032,Z 581.079,A -85,B 0,C 180,E1 1869.962,E2 1869.962} C_VEL
LIN {X 0,Y 585.619,Z 595.238,A -85,B 0,C 180,E1 1870.627,E2 1870.627} C_VEL
LIN {X 0,Y 585.225,Z 626.001,A -85,B 0,C 180,E1 1872.39,E2 1872.39} C_VEL
LIN {X 0,Y 584.82,Z 653.914,A -85,B 0,C 180,E1 1874.666,E2 1874.666} C_VEL
LIN {X 0,Y 584.427,Z 677.373,A -85,B 0,C 180,E1 1877.324,E2 1877.324} C_VEL
LIN {X 0,Y 584.247,Z 696.263,A -85,B 0,C 180,E1 1880.337,E2 1880.337} C_VEL
LIN {X 0,Y 584.136,Z 708.2,A -85,B 0,C 180,E1 1883.095,E2 1883.095} C_VEL
LIN {X 0,Y 584.174,Z 716.708,A -85,B 0,C 180,E1 1886.299,E2 1886.299} C_VEL
LIN {X 0,Y 584.175,Z 719.452,A -85,B 0,C 180,E1 1888.521,E2 1888.521} C_VEL
LIN {X 0,Y 584.135,Z 719.389,A -85,B 0,C 180,E1 1891.481,E2 1891.481} C_VEL
LIN {X 0,Y 584.18,Z 715.006,A -85,B 0,C 180,E1 1894.445,E2 1894.445} C_VEL
LIN {X 0,Y 584.296,Z 704.482,A -85,B 0,C 180,E1 1897.793,E2 1897.793} C_VEL
LIN {X 0,Y 584.422,Z 688.039,A -85,B 0,C 180,E1 1901.021,E2 1901.021} C_VEL
LIN {X 0,Y 584.709,Z 666.828,A -85,B 0,C 180,E1 1903.888,E2 1903.888} C_VEL
LIN {X 0,Y 585.034,Z 641.042,A -85,B 0,C 180,E1 1906.387,E2 1906.387} C_VEL
LIN {X 0,Y 585.447,Z 611.974,A -85,B 0,C 180,E1 1908.406,E2 1908.406} C_VEL
LIN {X 0,Y 585.034,Z 584.92,A -85,B 0,C 180,E1 1909.757,E2 1909.757} C_VEL
LIN {X 0,Y 584.129,Z 580.66,A -85,B 0,C 180,E1 1910.002,E2 1910.002} C_VEL
LIN {X 0,Y 583.772,Z 580.66,A -85,B 0,C 180,E1 1916.068,E2 1916.068} C_VEL
LIN {X 0,Y 583.594,Z 580.66,A -85,B 0,C 180,E1 1921.444,E2 1921.444} C_VEL
LIN {X 0,Y 583.832,Z 580.66,A -85,B 0,C 180,E1 1926.763,E2 1926.763} C_VEL
LIN {X 0,Y 583.553,Z 580.66,A -85,B 0,C 180,E1 1932.246,E2 1932.246} C_VEL
LIN {X 0,Y 583.708,Z 580.66,A -85,B 0,C 180,E1 1937.775,E2 1937.775} C_VEL
LIN {X 0,Y 583.725,Z 580.66,A -85,B 0,C 180,E1 1943.525,E2 1943.525} C_VEL
LIN {X 0,Y 583.617,Z 580.66,A -85,B 0,C 180,E1 1948.867,E2 1948.867} C_VEL
LIN {X 0,Y 583.794,Z 580.66,A -85,B 0,C 180,E1 1954.777,E2 1954.777} C_VEL
LIN {X 0,Y 583.91,Z 580.66,A -85,B 0,C 180,E1 1960.374,E2 1960.374} C_VEL
LIN {X 0,Y 583.6,Z 580.66,A -85,B 0,C 180,E1 1965.019,E2 1965.019} C_VEL
LIN {X 0,Y 583.731,Z 580.66,A -85,B 0,C 180,E1 1971.081,E2 1971.081} C_VEL
LIN {X 0,Y 583.839,Z 580.66,A -85,B 0,C 180,E1 1975.556,E2 1975.556} C_VEL
LIN {X 0,Y 583.896,Z 580.66,A -85,B 0,C 180,E1 1980.003,E2 1980.003} C_VEL
LIN {X 0,Y 583.903,Z 580.66,A -85,B 0,C 180,E1 1984.449,E2 1984.449} C_VEL
LIN {X 0,Y 583.743,Z 580.66,A -85,B 0,C 180,E1 1985.892,E2 1985.892} C_VEL
LIN {X 0,Y 579.965,Z 580.66,A -85,B 0,C 180,E1 1987.571,E2 1987.571} C_VEL
LIN {X 0,Y 575.971,Z 580.66,A -85,B 0,C 180,E1 1989.272,E2 1989.272} C_VEL
LIN {X 0,Y 575.916,Z 580.66,A -85,B 0,C 180,E1 1994.203,E2 1994.203} C_VEL
LIN {X 0,Y 575.833,Z 580.66,A -85,B 0,C 180,E1 1999.919,E2 1999.919} C_VEL
LIN {X 0,Y 575.732,Z 580.66,A -85,B 0,C 180,E1 2004.795,E2 2004.795} C_VEL
LIN {X 0,Y 575.664,Z 580.66,A -85,B 0,C 180,E1 2010.116,E2 2010.116} C_VEL
LIN {X 0,Y 575.688,Z 580.66,A -85,B 0,C 180,E1 2015.216,E2 2015.216} C_VEL
LIN {X 0,Y 575.646,Z 580.66,A -85,B 0,C 180,E1 2020.945,E2 2020.945} C_VEL
LIN {X 0,Y 575.8,Z 580.66,A -85,B 0,C 180,E1 2027.204,E2 2027.204} C_VEL
LIN {X 0,Y 575.839,Z 580.66,A -85,B 0,C 180,E1 2032.936,E2 2032.936} C_VEL
LIN {X 0,Y 575.756,Z 580.66,A -85,B 0,C 180,E1 2038.387,E2 2038.387} C_VEL
LIN {X 0,Y 575.912,Z 580.66,A -85,B 0,C 180,E1 2042.684,E2 2042.684} C_VEL
LIN {X 0,Y 579.776,Z 594.461,A -85,B 0,C 180,E1 2043.075,E2 2043.075} C_VEL
LIN {X 0,Y 579.779,Z 666.717,A -85,B 0,C 180,E1 2044.179,E2 2044.179} C_VEL
LIN {X 0,Y 579.239,Z 703.72,A -85,B 0,C 180,E1 2045.366,E2 2045.366} C_VEL
LIN {X 0,Y 578.556,Z 737.833,A -85,B 0,C 180,E1 2047.064,E2 2047.064} C_VEL
LIN {X 0,Y 577.85,Z 770.605,A -85,B 0,C 180,E1 2049.358,E2 2049.358} C_VEL
LIN {X 0,Y 577.207,Z 799.38,A -85,B 0,C 180,E1 2052.092,E2 2052.092} C_VEL
LIN {X 0,Y 576.675,Z 824.136,A -85,B 0,C 180,E1 2055.24,E2 2055.24} C_VEL
LIN {X 0,Y 576.375,Z 843.445,A -85,B 0,C 180,E1 2058.582,E2 2058.582} C_VEL
LIN {X 0,Y 576.262,Z 857.536,A -85,B 0,C 180,E1 2062.097,E2 2062.097} C_VEL
LIN {X 0,Y 576.152,Z 865.991,A -85,B 0,C 180,E1 2065.492,E2 2065.492} C_VEL
LIN {X 0,Y 576.162,Z 869.511,A -85,B 0,C 180,E1 2068.498,E2 2068.498} C_VEL
LIN {X 0,Y 576.311,Z 869.513,A -85,B 0,C 180,E1 2071.499,E2 2071.499} C_VEL
LIN {X 0,Y 576.226,Z 865.995,A -85,B 0,C 180,E1 2074.504,E2 2074.504} C_VEL
LIN {X 0,Y 576.332,Z 856.279,A -85,B 0,C 180,E1 2078.278,E2 2078.278} C_VEL
LIN {X 0,Y 576.395,Z 841.085,A -85,B 0,C 180,E1 2081.881,E2 2081.881} C_VEL
LIN {X 0,Y 576.768,Z 821.344,A -85,B 0,C 180,E1 2085.165,E2 2085.165} C_VEL
LIN {X 0,Y 577.271,Z 795.967,A -85,B 0,C 180,E1 2088.279,E2 2088.279} C_VEL
LIN {X 0,Y 577.946,Z 766.141,A -85,B 0,C 180,E1 2090.997,E2 2090.997} C_VEL
LIN {X 0,Y 578.724,Z 732.557,A -85,B 0,C 180,E1 2093.245,E2 2093.245} C_VEL
LIN {X 0,Y 579.387,Z 697.398,A -85,B 0,C 180,E1 2094.881,E2 2094.881} C_VEL
LIN {X 0,Y 579.911,Z 661.407,A -85,B 0,C 180,E1 2095.93,E2 2095.93} C_VEL
LIN {X 0,Y 578.829,Z 588.45,A -85,B 0,C 180,E1 2097.054,E2 2097.054} C_VEL
LIN {X 0,Y 576.164,Z 580.66,A -85,B 0,C 180,E1 2097.349,E2 2097.349} C_VEL
LIN {X 0,Y 575.876,Z 580.66,A -85,B 0,C 180,E1 2103.382,E2 2103.382} C_VEL
LIN {X 0,Y 575.685,Z 580.66,A -85,B 0,C 180,E1 2108.979,E2 2108.979} C_VEL
LIN {X 0,Y 575.768,Z 580.66,A -85,B 0,C 180,E1 2115.037,E2 2115.037} C_VEL
LIN {X 0,Y 575.758,Z 580.66,A -85,B 0,C 180,E1 2121.023,E2 2121.023} C_VEL
LIN {X 0,Y 575.671,Z 580.66,A -85,B 0,C 180,E1 2126.601,E2 2126.601} C_VEL
LIN {X 0,Y 575.738,Z 580.66,A -85,B 0,C 180,E1 2131.85,E2 2131.85} C_VEL
LIN {X 0,Y 575.678,Z 580.66,A -85,B 0,C 180,E1 2136.846,E2 2136.846} C_VEL
LIN {X 0,Y 575.937,Z 580.66,A -85,B 0,C 180,E1 2141.674,E2 2141.674} C_VEL
LIN {X 0,Y 575.73,Z 580.66,A -85,B 0,C 180,E1 2147.895,E2 2147.895} C_VEL
LIN {X 0,Y 576.191,Z 580.66,A -85,B 0,C 180,E1 2153.985,E2 2153.985} C_VEL
LIN {X 0,Y 575.969,Z 580.66,A -85,B 0,C 180,E1 2159.997,E2 2159.997} C_VEL
LIN {X 0,Y 576.025,Z 580.66,A -85,B 0,C 180,E1 2164.504,E2 2164.504} C_VEL
LIN {X 0,Y 575.997,Z 580.66,A -85,B 0,C 180,E1 2169.04,E2 2169.04} C_VEL
LIN {X 0,Y 575.884,Z 580.66,A -85,B 0,C 180,E1 2174.201,E2 2174.201} C_VEL
LIN {X 0,Y 575.831,Z 580.66,A -85,B 0,C 180,E1 2179.913,E2 2179.913} C_VEL
LIN {X 0,Y 575.724,Z 580.66,A -85,B 0,C 180,E1 2184.789,E2 2184.789} C_VEL
LIN {X 0,Y 575.659,Z 580.66,A -85,B 0,C 180,E1 2190.12,E2 2190.12} C_VEL
LIN {X 0,Y 575.675,Z 580.66,A -85,B 0,C 180,E1 2195.21,E2 2195.21} C_VEL
LIN {X 0,Y 575.614,Z 580.66,A -85,B 0,C 180,E1 2200.941,E2 2200.941} C_VEL
LIN {X 0,Y 575.806,Z 580.66,A -85,B 0,C 180,E1 2207.054,E2 2207.054} C_VEL
LIN {X 0,Y 575.817,Z 580.66,A -85,B 0,C 180,E1 2212.937,E2 2212.937} C_VEL
LIN {X 0,Y 575.715,Z 580.66,A -85,B 0,C 180,E1 2218.388,E2 2218.388} C_VEL
LIN {X 0,Y 575.805,Z 580.66,A -85,B 0,C 180,E1 2223.547,E2 2223.547} C_VEL
LIN {X 0,Y 576.112,Z 580.66,A -85,B 0,C 180,E1 2229.646,E2 2229.646} C_VEL
LIN {X 0,Y 578.105,Z 595.825,A -85,B 0,C 180,E1 2230.393,E2 2230.393} C_VEL
LIN {X 0,Y 577.58,Z 626.917,A -85,B 0,C 180,E1 2232.215,E2 2232.215} C_VEL
LIN {X 0,Y 577.085,Z 653.906,A -85,B 0,C 180,E1 2234.456,E2 2234.456} C_VEL
LIN {X 0,Y 576.62,Z 677.367,A -85,B 0,C 180,E1 2237.149,E2 2237.149} C_VEL
LIN {X 0,Y 576.408,Z 696.261,A -85,B 0,C 180,E1 2240.204,E2 2240.204} C_VEL
LIN {X 0,Y 576.232,Z 709.024,A -85,B 0,C 180,E1 2243.234,E2 2243.234} C_VEL
LIN {X 0,Y 576.299,Z 716.707,A -85,B 0,C 180,E1 2246.248,E2 2246.248} C_VEL
LIN {X 0,Y 576.272,Z 719.453,A -85,B 0,C 180,E1 2248.501,E2 2248.501} C_VEL
LIN {X 0,Y 576.233,Z 719.389,A -85,B 0,C 180,E1 2251.502,E2 2251.502} C_VEL
LIN {X 0,Y 576.285,Z 715.006,A -85,B 0,C 180,E1 2254.507,E2 2254.507} C_VEL
LIN {X 0,Y 576.44,Z 704.484,A -85,B 0,C 180,E1 2257.9,E2 2257.9} C_VEL
LIN {X 0,Y 576.613,Z 688.178,A -85,B 0,C 180,E1 2261.15,E2 2261.15} C_VEL
LIN {X 0,Y 576.944,Z 666.495,A -85,B 0,C 180,E1 2264.119,E2 2264.119} C_VEL
LIN {X 0,Y 577.347,Z 641.047,A -85,B 0,C 180,E1 2266.611,E2 2266.611} C_VEL
LIN {X 0,Y 577.891,Z 611.99,A -85,B 0,C 180,E1 2268.656,E2 2268.656} C_VEL
LIN {X 0,Y 577.368,Z 586.01,A -85,B 0,C 180,E1 2269.986,E2 2269.986} C_VEL
LIN {X 0,Y 576.166,Z 580.66,A -85,B 0,C 180,E1 2270.265,E2 2270.265} C_VEL
LIN {X 0,Y 575.772,Z 580.66,A -85,B 0,C 180,E1 2276.458,E2 2276.458} C_VEL
LIN {X 0,Y 575.686,Z 580.66,A -85,B 0,C 180,E1 2281.617,E2 2281.617} C_VEL
LIN {X 0,Y 575.92,Z 580.66,A -85,B 0,C 180,E1 2287.058,E2 2287.058} C_VEL
LIN {X 0,Y 575.648,Z 580.66,A -85,B 0,C 180,E1 2292.965,E2 2292.965} C_VEL
LIN {X 0,Y 575.775,Z 580.66,A -85,B 0,C 180,E1 2299.073,E2 2299.073} C_VEL
LIN {X 0,Y 575.683,Z 580.66,A -85,B 0,C 180,E1 2304.79,E2 2304.79} C_VEL
LIN {X 0,Y 575.691,Z 580.66,A -85,B 0,C 180,E1 2310.137,E2 2310.137} C_VEL
LIN {X 0,Y 575.841,Z 580.66,A -85,B 0,C 180,E1 2315.216,E2 2315.216} C_VEL
LIN {X 0,Y 575.995,Z 580.66,A -85,B 0,C 180,E1 2320.579,E2 2320.579} C_VEL
LIN {X 0,Y 575.591,Z 580.66,A -85,B 0,C 180,E1 2325.925,E2 2325.925} C_VEL
LIN {X 0,Y 575.854,Z 580.66,A -85,B 0,C 180,E1 2330.958,E2 2330.958} C_VEL
LIN {X 0,Y 575.944,Z 580.66,A -85,B 0,C 180,E1 2335.495,E2 2335.495} C_VEL
LIN {X 0,Y 575.995,Z 580.66,A -85,B 0,C 180,E1 2340.003,E2 2340.003} C_VEL
LIN {X 0,Y 575.881,Z 580.66,A -85,B 0,C 180,E1 2345.32,E2 2345.32} C_VEL
LIN {X 0,Y 575.971,Z 580.66,A -85,B 0,C 180,E1 2349.272,E2 2349.272} C_VEL
LIN {X 0,Y 571.924,Z 580.66,A -85,B 0,C 180,E1 2350.967,E2 2350.967} C_VEL
LIN {X 0,Y 568.026,Z 580.66,A -85,B 0,C 180,E1 2352.686,E2 2352.686} C_VEL
LIN {X 0,Y 568.021,Z 580.66,A -85,B 0,C 180,E1 2358.591,E2 2358.591} C_VEL
LIN {X 0,Y 567.929,Z 580.66,A -85,B 0,C 180,E1 2363.489,E2 2363.489} C_VEL
LIN {X 0,Y 567.836,Z 580.66,A -85,B 0,C 180,E1 2368.725,E2 2368.725} C_VEL
LIN {X 0,Y 567.788,Z 580.66,A -85,B 0,C 180,E1 2374.527,E2 2374.527} C_VEL
LIN {X 0,Y 567.75,Z 580.66,A -85,B 0,C 180,E1 2379.634,E2 2379.634} C_VEL
LIN {X 0,Y 567.781,Z 580.66,A -85,B 0,C 180,E1 2385.854,E2 2385.854} C_VEL
LIN {X 0,Y 567.852,Z 580.66,A -85,B 0,C 180,E1 2390.41,E2 2390.41} C_VEL
LIN {X 0,Y 567.73,Z 580.66,A -85,B 0,C 180,E1 2395.481,E2 2395.481} C_VEL
LIN {X 0,Y 567.861,Z 580.66,A -85,B 0,C 180,E1 2401.269,E2 2401.269} C_VEL
LIN {X 0,Y 567.986,Z 580.66,A -85,B 0,C 180,E1 2402.273,E2 2402.273} C_VEL
LIN {X 0,Y 572.775,Z 596.071,A -85,B 0,C 180,E1 2402.741,E2 2402.741} C_VEL
LIN {X 0,Y 572.672,Z 667.124,A -85,B 0,C 180,E1 2403.845,E2 2403.845} C_VEL
LIN {X 0,Y 571.962,Z 703.718,A -85,B 0,C 180,E1 2405.031,E2 2405.031} C_VEL
LIN {X 0,Y 571.156,Z 738.816,A -85,B 0,C 180,E1 2406.81,E2 2406.81} C_VEL
LIN {X 0,Y 570.302,Z 771.822,A -85,B 0,C 180,E1 2409.173,E2 2409.173} C_VEL
LIN {X 0,Y 569.51,Z 800.257,A -85,B 0,C 180,E1 2411.942,E2 2411.942} C_VEL
LIN {X 0,Y 568.909,Z 824.132,A -85,B 0,C 180,E1 2415.033,E2 2415.033} C_VEL
LIN {X 0,Y 568.54,Z 843.905,A -85,B 0,C 180,E1 2418.518,E2 2418.518} C_VEL
LIN {X 0,Y 568.394,Z 857.536,A -85,B 0,C 180,E1 2421.987,E2 2421.987} C_VEL
LIN {X 0,Y 568.275,Z 865.99,A -85,B 0,C 180,E1 2425.43,E2 2425.43} C_VEL
LIN {X 0,Y 568.288,Z 869.511,A -85,B 0,C 180,E1 2428.477,E2 2428.477} C_VEL
LIN {X 0,Y 568.427,Z 869.513,A -85,B 0,C 180,E1 2431.52,E2 2431.52} C_VEL
LIN {X 0,Y 568.33,Z 865.995,A -85,B 0,C 180,E1 2434.567,E2 2434.567} C_VEL
LIN {X 0,Y 568.441,Z 856.279,A -85,B 0,C 180,E1 2438.394,E2 2438.394} C_VEL
LIN {X 0,Y 568.55,Z 841.923,A -85,B 0,C 180,E1 2441.881,E2 2441.881} C_VEL
LIN {X 0,Y 568.964,Z 822.679,A -85,B 0,C 180,E1 2445.181,E2 2445.181} C_VEL
LIN {X 0,Y 569.578,Z 797.584,A -85,B 0,C 180,E1 2448.361,E2 2448.361} C_VEL
LIN {X 0,Y 570.394,Z 768.138,A -85,B 0,C 180,E1 2451.126,E2 2451.126} C_VEL
LIN {X 0,Y 571.255,Z 736.296,A -85,B 0,C 180,E1 2453.34,E2 2453.34} C_VEL
LIN {X 0,Y 572.065,Z 700.517,A -85,B 0,C 180,E1 2455.102,E2 2455.102} C_VEL
LIN {X 0,Y 572.768,Z 663.431,A -85,B 0,C 180,E1 2456.234,E2 2456.234} C_VEL
LIN {X 0,Y 571.742,Z 590.501,A -85,B 0,C 180,E1 2457.389,E2 2457.389} C_VEL
LIN {X 0,Y 568.144,Z 580.66,A -85,B 0,C 180,E1 2457.779,E2 2457.779} C_VEL
LIN {X 0,Y 567.862,Z 580.66,A -85,B 0,C 180,E1 2463.917,E2 2463.917} C_VEL
LIN {X 0,Y 567.741,Z 580.66,A -85,B 0,C 180,E1 2469.631,E2 2469.631} C_VEL
LIN {X 0,Y 567.798,Z 580.66,A -85,B 0,C 180,E1 2475.848,E2 2475.848} C_VEL
LIN {X 0,Y 567.841,Z 580.66,A -85,B 0,C 180,E1 2480.407,E2 2480.407} C_VEL
LIN {X 0,Y 567.72,Z 580.66,A -85,B 0,C 180,E1 2485.478,E2 2485.478} C_VEL
LIN {X 0,Y 567.789,Z 580.66,A -85,B 0,C 180,E1 2491.278,E2 2491.278} C_VEL
LIN {X 0,Y 567.8,Z 580.66,A -85,B 0,C 180,E1 2496.506,E2 2496.506} C_VEL
LIN {X 0,Y 568.048,Z 580.66,A -85,B 0,C 180,E1 2501.41,E2 2501.41} C_VEL
LIN {X 0,Y 567.702,Z 580.66,A -85,B 0,C 180,E1 2506.157,E2 2506.157} C_VEL
LIN {X 0,Y 567.962,Z 580.66,A -85,B 0,C 180,E1 2510.825,E2 2510.825} C_VEL
LIN {X 0,Y 568.019,Z 580.66,A -85,B 0,C 180,E1 2515.426,E2 2515.426} C_VEL
LIN {X 0,Y 568.094,Z 580.66,A -85,B 0,C 180,E1 2519.997,E2 2519.997} C_VEL
LIN {X 0,Y 568.112,Z 580.66,A -85,B 0,C 180,E1 2524.567,E2 2524.567} C_VEL
LIN {X 0,Y 568.064,Z 580.66,A -85,B 0,C 180,E1 2529.167,E2 2529.167} C_VEL
LIN {X 0,Y 568.071,Z 580.66,A -85,B 0,C 180,E1 2533.828,E2 2533.828} C_VEL
LIN {X 0,Y 568.037,Z 580.66,A -85,B 0,C 180,E1 2538.584,E2 2538.584} C_VEL
LIN {X 0,Y 567.909,Z 580.66,A -85,B 0,C 180,E1 2543.483,E2 2543.483} C_VEL
LIN {X 0,Y 567.819,Z 580.66,A -85,B 0,C 180,E1 2548.727,E2 2548.727} C_VEL
LIN {X 0,Y 567.775,Z 580.66,A -85,B 0,C 180,E1 2554.53,E2 2554.53} C_VEL
LIN {X 0,Y 567.704,Z 580.66,A -85,B 0,C 180,E1 2559.63,E2 2559.63} C_VEL
LIN {X 0,Y 567.784,Z 580.66,A -85,B 0,C 180,E1 2565.845,E2 2565.845} C_VEL
LIN {X 0,Y 567.824,Z 580.66,A -85,B 0,C 180,E1 2570.404,E2 2570.404} C_VEL
LIN {X 0,Y 567.718,Z 580.66,A -85,B 0,C 180,E1 2575.473,E2 2575.473} C_VEL
LIN {X 0,Y 567.764,Z 580.66,A -85,B 0,C 180,E1 2581.276,E2 2581.276} C_VEL
LIN {X 0,Y 567.873,Z 580.66,A -85,B 0,C 180,E1 2586.513,E2 2586.513} C_VEL
LIN {X 0,Y 568.157,Z 580.888,A -85,B 0,C 180,E1 2589.371,E2 2589.371} C_VEL
LIN {X 0,Y 570.647,Z 595.816,A -85,B 0,C 180,E1 2590.126,E2 2590.126} C_VEL
LIN {X 0,Y 569.992,Z 625.85,A -85,B 0,C 180,E1 2591.894,E2 2591.894} C_VEL
LIN {X 0,Y 569.321,Z 653.897,A -85,B 0,C 180,E1 2594.238,E2 2594.238} C_VEL
LIN {X 0,Y 568.841,Z 677.361,A -85,B 0,C 180,E1 2596.971,E2 2596.971} C_VEL
LIN {X 0,Y 568.54,Z 696.258,A -85,B 0,C 180,E1 2600.067,E2 2600.067} C_VEL
LIN {X 0,Y 568.352,Z 709.022,A -85,B 0,C 180,E1 2603.14,E2 2603.14} C_VEL
LIN {X 0,Y 568.407,Z 716.705,A -85,B 0,C 180,E1 2606.196,E2 2606.196} C_VEL
LIN {X 0,Y 568.387,Z 719.452,A -85,B 0,C 180,E1 2608.48,E2 2608.48} C_VEL
LIN {X 0,Y 568.351,Z 719.389,A -85,B 0,C 180,E1 2611.523,E2 2611.523} C_VEL
LIN {X 0,Y 568.471,Z 713.709,A -85,B 0,C 180,E1 2615.123,E2 2615.123} C_VEL
LIN {X 0,Y 568.535,Z 702.958,A -85,B 0,C 180,E1 2618.395,E2 2618.395} C_VEL
LIN {X 0,Y 568.803,Z 686.704,A -85,B 0,C 180,E1 2621.544,E2 2621.544} C_VEL
LIN {X 0,Y 569.175,Z 665.265,A -85,B 0,C 180,E1 2624.455,E2 2624.455} C_VEL
LIN {X 0,Y 569.691,Z 639.906,A -85,B 0,C 180,E1 2626.94,E2 2626.94} C_VEL
LIN {X 0,Y 570.352,Z 610.303,A -85,B 0,C 180,E1 2629.012,E2 2629.012} C_VEL
LIN {X 0,Y 569.983,Z 588.149,A -85,B 0,C 180,E1 2630.167,E2 2630.167} C_VEL
LIN {X 0,Y 568.192,Z 580.66,A -85,B 0,C 180,E1 2630.633,E2 2630.633} C_VEL
LIN {X 0,Y 567.801,Z 580.66,A -85,B 0,C 180,E1 2636.859,E2 2636.859} C_VEL
LIN {X 0,Y 567.731,Z 580.66,A -85,B 0,C 180,E1 2642.112,E2 2642.112} C_VEL
LIN {X 0,Y 567.991,Z 580.66,A -85,B 0,C 180,E1 2647.664,E2 2647.664} C_VEL
LIN {X 0,Y 567.702,Z 580.66,A -85,B 0,C 180,E1 2654.146,E2 2654.146} C_VEL
LIN {X 0,Y 567.801,Z 580.66,A -85,B 0,C 180,E1 2658.372,E2 2658.372} C_VEL
LIN {X 0,Y 567.823,Z 580.66,A -85,B 0,C 180,E1 2664.229,E2 2664.229} C_VEL
LIN {X 0,Y 567.785,Z 580.66,A -85,B 0,C 180,E1 2669.678,E2 2669.678} C_VEL
LIN {X 0,Y 567.886,Z 580.66,A -85,B 0,C 180,E1 2674.845,E2 2674.845} C_VEL
LIN {X 0,Y 568.021,Z 580.66,A -85,B 0,C 180,E1 2679.801,E2 2679.801} C_VEL
LIN {X 0,Y 567.845,Z 580.66,A -85,B 0,C 180,E1 2684.593,E2 2684.593} C_VEL
LIN {X 0,Y 567.946,Z 580.66,A -85,B 0,C 180,E1 2690.831,E2 2690.831} C_VEL
LIN {X 0,Y 568.053,Z 580.66,A -85,B 0,C 180,E1 2695.432,E2 2695.432} C_VEL
LIN {X 0,Y 568.119,Z 580.66,A -85,B 0,C 180,E1 2700.003,E2 2700.003} C_VEL
LIN {X 0,Y 568.077,Z 580.66,A -85,B 0,C 180,E1 2704.573,E2 2704.573} C_VEL
LIN {X 0,Y 568.075,Z 580.66,A -85,B 0,C 180,E1 2709.256,E2 2709.256} C_VEL
LIN {X 0,Y 568.026,Z 580.66,A -85,B 0,C 180,E1 2712.686,E2 2712.686} C_VEL
LIN {X 0,Y 565.443,Z 580.66,A -85,B 0,C 180,E1 2713.983,E2 2713.983} C_VEL
LIN {X 0,Y 560.042,Z 580.66,A -85,B 0,C 180,E1 2715.926,E2 2715.926} C_VEL
LIN {X 0,Y 559.951,Z 580.66,A -85,B 0,C 180,E1 2716.15,E2 2716.15} C_VEL
LIN {X 0,Y 559.986,Z 580.66,A -85,B 0,C 180,E1 2720.508,E2 2720.508} C_VEL
LIN {X 0,Y 559.873,Z 580.66,A -85,B 0,C 180,E1 2725.547,E2 2725.547} C_VEL
LIN {X 0,Y 559.862,Z 580.66,A -85,B 0,C 180,E1 2730.805,E2 2730.805} C_VEL
LIN {X 0,Y 559.801,Z 580.66,A -85,B 0,C 180,E1 2736.372,E2 2736.372} C_VEL
LIN {X 0,Y 559.763,Z 580.66,A -85,B 0,C 180,E1 2742.371,E2 2742.371} C_VEL
LIN {X 0,Y 559.892,Z 580.66,A -85,B 0,C 180,E1 2747.641,E2 2747.641} C_VEL
LIN {X 0,Y 559.949,Z 580.66,A -85,B 0,C 180,E1 2753.944,E2 2753.944} C_VEL
LIN {X 0,Y 559.977,Z 580.66,A -85,B 0,C 180,E1 2759.575,E2 2759.575} C_VEL
LIN {X 0,Y 560.048,Z 580.66,A -85,B 0,C 180,E1 2761.845,E2 2761.845} C_VEL
LIN {X 0,Y 565.732,Z 596.402,A -85,B 0,C 180,E1 2762.378,E2 2762.378} C_VEL
LIN {X 0,Y 565.559,Z 667.428,A -85,B 0,C 180,E1 2763.499,E2 2763.499} C_VEL
LIN {X 0,Y 564.763,Z 703.715,A -85,B 0,C 180,E1 2764.691,E2 2764.691} C_VEL
LIN {X 0,Y 563.797,Z 738.425,A -85,B 0,C 180,E1 2766.464,E2 2766.464} C_VEL
LIN {X 0,Y 562.77,Z 771.822,A -85,B 0,C 180,E1 2768.881,E2 2768.881} C_VEL
LIN {X 0,Y 561.81,Z 801.026,A -85,B 0,C 180,E1 2771.775,E2 2771.775} C_VEL
LIN {X 0,Y 561.096,Z 825.596,A -85,B 0,C 180,E1 2775.041,E2 2775.041} C_VEL
LIN {X 0,Y 560.685,Z 843.902,A -85,B 0,C 180,E1 2778.354,E2 2778.354} C_VEL
LIN {X 0,Y 560.539,Z 857.536,A -85,B 0,C 180,E1 2781.874,E2 2781.874} C_VEL
LIN {X 0,Y 560.391,Z 865.99,A -85,B 0,C 180,E1 2785.365,E2 2785.365} C_VEL
LIN {X 0,Y 560.387,Z 869.511,A -85,B 0,C 180,E1 2788.456,E2 2788.456} C_VEL
LIN {X 0,Y 560.524,Z 869.513,A -85,B 0,C 180,E1 2791.541,E2 2791.541} C_VEL
LIN {X 0,Y 560.412,Z 865.369,A -85,B 0,C 180,E1 2794.968,E2 2794.968} C_VEL
LIN {X 0,Y 560.566,Z 856.279,A -85,B 0,C 180,E1 2798.512,E2 2798.512} C_VEL
LIN {X 0,Y 560.681,Z 841.989,A -85,B 0,C 180,E1 2802.037,E2 2802.037} C_VEL
LIN {X 0,Y 561.187,Z 822.368,A -85,B 0,C 180,E1 2805.443,E2 2805.443} C_VEL
LIN {X 0,Y 561.905,Z 797.27,A -85,B 0,C 180,E1 2808.657,E2 2808.657} C_VEL
LIN {X 0,Y 562.904,Z 766.894,A -85,B 0,C 180,E1 2811.524,E2 2811.524} C_VEL
LIN {X 0,Y 563.943,Z 734.271,A -85,B 0,C 180,E1 2813.786,E2 2813.786} C_VEL
LIN {X 0,Y 564.985,Z 698.115,A -85,B 0,C 180,E1 2815.533,E2 2815.533} C_VEL
LIN {X 0,Y 565.685,Z 663.431,A -85,B 0,C 180,E1 2816.588,E2 2816.588} C_VEL
LIN {X 0,Y 565.019,Z 593.327,A -85,B 0,C 180,E1 2817.703,E2 2817.703} C_VEL
LIN {X 0,Y 560.166,Z 580.66,A -85,B 0,C 180,E1 2818.202,E2 2818.202} C_VEL
LIN {X 0,Y 559.913,Z 580.66,A -85,B 0,C 180,E1 2824.465,E2 2824.465} C_VEL
LIN {X 0,Y 559.742,Z 580.66,A -85,B 0,C 180,E1 2830.312,E2 2830.312} C_VEL
LIN {X 0,Y 559.844,Z 580.66,A -85,B 0,C 180,E1 2835.51,E2 2835.51} C_VEL
LIN {X 0,Y 559.891,Z 580.66,A -85,B 0,C 180,E1 2841.401,E2 2841.401} C_VEL
LIN {X 0,Y 559.797,Z 580.66,A -85,B 0,C 180,E1 2846.676,E2 2846.676} C_VEL
LIN {X 0,Y 559.871,Z 580.66,A -85,B 0,C 180,E1 2850.978,E2 2850.978} C_VEL
LIN {X 0,Y 559.916,Z 580.66,A -85,B 0,C 180,E1 2856.383,E2 2856.383} C_VEL
LIN {X 0,Y 560.111,Z 580.66,A -85,B 0,C 180,E1 2861.137,E2 2861.137} C_VEL
LIN {X 0,Y 559.819,Z 580.66,A -85,B 0,C 180,E1 2866.003,E2 2866.003} C_VEL
LIN {X 0,Y 560.059,Z 580.66,A -85,B 0,C 180,E1 2870.695,E2 2870.695} C_VEL
LIN {X 0,Y 560.143,Z 580.66,A -85,B 0,C 180,E1 2875.362,E2 2875.362} C_VEL
LIN {X 0,Y 560.193,Z 580.66,A -85,B 0,C 180,E1 2879.997,E2 2879.997} C_VEL
LIN {X 0,Y 560.206,Z 580.66,A -85,B 0,C 180,E1 2884.745,E2 2884.745} C_VEL
LIN {X 0,Y 560.167,Z 580.66,A -85,B 0,C 180,E1 2889.298,E2 2889.298} C_VEL
LIN {X 0,Y 560.103,Z 580.66,A -85,B 0,C 180,E1 2894.113,E2 2894.113} C_VEL
LIN {X 0,Y 560.021,Z 580.66,A -85,B 0,C 180,E1 2899.436,E2 2899.436} C_VEL
LIN {X 0,Y 559.945,Z 580.66,A -85,B 0,C 180,E1 2903.838,E2 2903.838} C_VEL
LIN {X 0,Y 559.881,Z 580.66,A -85,B 0,C 180,E1 2909.015,E2 2909.015} C_VEL
LIN {X 0,Y 559.893,Z 580.66,A -85,B 0,C 180,E1 2914.463,E2 2914.463} C_VEL
LIN {X 0,Y 559.709,Z 580.66,A -85,B 0,C 180,E1 2920.311,E2 2920.311} C_VEL
LIN {X 0,Y 559.834,Z 580.66,A -85,B 0,C 180,E1 2925.513,E2 2925.513} C_VEL
LIN {X 0,Y 559.875,Z 580.66,A -85,B 0,C 180,E1 2931.398,E2 2931.398} C_VEL
LIN {X 0,Y 559.787,Z 580.66,A -85,B 0,C 180,E1 2936.671,E2 2936.671} C_VEL
LIN {X 0,Y 559.845,Z 580.66,A -85,B 0,C 180,E1 2940.98,E2 2940.98} C_VEL
LIN {X 0,Y 559.957,Z 580.66,A -85,B 0,C 180,E1 2946.364,E2 2946.364} C_VEL
LIN {X 0,Y 560.207,Z 581.387,A -85,B 0,C 180,E1 2949.086,E2 2949.086} C_VEL
LIN {X 0,Y 563.135,Z 597.245,A -85,B 0,C 180,E1 2949.919,E2 2949.919} C_VEL
LIN {X 0,Y 562.354,Z 628.114,A -85,B 0,C 180,E1 2951.806,E2 2951.806} C_VEL
LIN {X 0,Y 561.579,Z 655.806,A -85,B 0,C 180,E1 2954.215,E2 2954.215} C_VEL
LIN {X 0,Y 561.014,Z 678.781,A -85,B 0,C 180,E1 2956.983,E2 2956.983} C_VEL
LIN {X 0,Y 560.696,Z 696.254,A -85,B 0,C 180,E1 2959.927,E2 2959.927} C_VEL
LIN {X 0,Y 560.484,Z 709.02,A -85,B 0,C 180,E1 2963.043,E2 2963.043} C_VEL
LIN {X 0,Y 560.522,Z 716.703,A -85,B 0,C 180,E1 2966.142,E2 2966.142} C_VEL
LIN {X 0,Y 560.483,Z 719.452,A -85,B 0,C 180,E1 2968.459,E2 2968.459} C_VEL
LIN {X 0,Y 560.449,Z 719.389,A -85,B 0,C 180,E1 2971.544,E2 2971.544} C_VEL
LIN {X 0,Y 560.508,Z 715.007,A -85,B 0,C 180,E1 2974.634,E2 2974.634} C_VEL
LIN {X 0,Y 560.663,Z 704.489,A -85,B 0,C 180,E1 2978.124,E2 2978.124} C_VEL
LIN {X 0,Y 560.931,Z 688.557,A -85,B 0,C 180,E1 2981.405,E2 2981.405} C_VEL
LIN {X 0,Y 561.387,Z 666.762,A -85,B 0,C 180,E1 2984.487,E2 2984.487} C_VEL
LIN {X 0,Y 562.015,Z 641.057,A -85,B 0,C 180,E1 2987.078,E2 2987.078} C_VEL
LIN {X 0,Y 562.801,Z 610.993,A -85,B 0,C 180,E1 2989.236,E2 2989.236} C_VEL
LIN {X 0,Y 562.292,Z 588.994,A -85,B 0,C 180,E1 2990.419,E2 2990.419} C_VEL
LIN {X 0,Y 560.202,Z 580.66,A -85,B 0,C 180,E1 2990.917,E2 2990.917} C_VEL
LIN {X 0,Y 559.836,Z 580.66,A -85,B 0,C 180,E1 2997.272,E2 2997.272} C_VEL
LIN {X 0,Y 559.762,Z 580.66,A -85,B 0,C 180,E1 3002.626,E2 3002.626} C_VEL
LIN {X 0,Y 559.975,Z 580.66,A -85,B 0,C 180,E1 3008.3,E2 3008.3} C_VEL
LIN {X 0,Y 559.771,Z 580.66,A -85,B 0,C 180,E1 3014.497,E2 3014.497} C_VEL
LIN {X 0,Y 559.835,Z 580.66,A -85,B 0,C 180,E1 3019.7,E2 3019.7} C_VEL
LIN {X 0,Y 559.815,Z 580.66,A -85,B 0,C 180,E1 3025.531,E2 3025.531} C_VEL
LIN {X 0,Y 559.814,Z 580.66,A -85,B 0,C 180,E1 3030.981,E2 3030.981} C_VEL
LIN {X 0,Y 559.893,Z 580.66,A -85,B 0,C 180,E1 3036.395,E2 3036.395} C_VEL
LIN {X 0,Y 560.14,Z 580.66,A -85,B 0,C 180,E1 3041.144,E2 3041.144} C_VEL
LIN {X 0,Y 559.79,Z 580.66,A -85,B 0,C 180,E1 3046.025,E2 3046.025} C_VEL
LIN {X 0,Y 560.041,Z 580.66,A -85,B 0,C 180,E1 3050.7,E2 3050.7} C_VEL
LIN {X 0,Y 560.163,Z 580.66,A -85,B 0,C 180,E1 3055.368,E2 3055.368} C_VEL
LIN {X 0,Y 560.217,Z 580.66,A -85,B 0,C 180,E1 3060.003,E2 3060.003} C_VEL
LIN {X 0,Y 560.173,Z 580.66,A -85,B 0,C 180,E1 3064.673,E2 3064.673} C_VEL
LIN {X 0,Y 560.176,Z 580.66,A -85,B 0,C 180,E1 3069.303,E2 3069.303} C_VEL
LIN {X 0,Y 560.151,Z 580.66,A -85,B 0,C 180,E1 3074.122,E2 3074.122} C_VEL
LIN {X 0,Y 559.951,Z 580.66,A -85,B 0,C 180,E1 3076.15,E2 3076.15} C_VEL
LIN {X 0,Y 558.73,Z 580.66,A -85,B 0,C 180,E1 3077.034,E2 3077.034} C_VEL
LIN {X 0,Y 552.069,Z 580.66,A -85,B 0,C 180,E1 3079.666,E2 3079.666} C_VEL
LIN {X 0,Y 551.976,Z 580.66,A -85,B 0,C 180,E1 3085.56,E2 3085.56} C_VEL
LIN {X 0,Y 551.913,Z 580.66,A -85,B 0,C 180,E1 3091.298,E2 3091.298} C_VEL
LIN {X 0,Y 551.814,Z 580.66,A -85,B 0,C 180,E1 3096.985,E2 3096.985} C_VEL
LIN {X 0,Y 551.847,Z 580.66,A -85,B 0,C 180,E1 3103.126,E2 3103.126} C_VEL
LIN {X 0,Y 552.001,Z 580.66,A -85,B 0,C 180,E1 3108.999,E2 3108.999} C_VEL
LIN {X 0,Y 551.956,Z 580.66,A -85,B 0,C 180,E1 3115.1,E2 3115.1} C_VEL
LIN {X 0,Y 552.089,Z 580.781,A -85,B 0,C 180,E1 3121.408,E2 3121.408} C_VEL
LIN {X 0,Y 558.802,Z 598.634,A -85,B 0,C 180,E1 3122.037,E2 3122.037} C_VEL
LIN {X 0,Y 558.494,Z 667.461,A -85,B 0,C 180,E1 3123.138,E2 3123.138} C_VEL
LIN {X 0,Y 557.58,Z 703.712,A -85,B 0,C 180,E1 3124.341,E2 3124.341} C_VEL
LIN {X 0,Y 556.485,Z 737.844,A -85,B 0,C 180,E1 3126.1,E2 3126.1} C_VEL
LIN {X 0,Y 555.29,Z 770.603,A -85,B 0,C 180,E1 3128.478,E2 3128.478} C_VEL
LIN {X 0,Y 554.205,Z 799.543,A -85,B 0,C 180,E1 3131.341,E2 3131.341} C_VEL
LIN {X 0,Y 553.439,Z 823.229,A -85,B 0,C 180,E1 3134.466,E2 3134.466} C_VEL
LIN {X 0,Y 552.907,Z 841.975,A -85,B 0,C 180,E1 3137.788,E2 3137.788} C_VEL
LIN {X 0,Y 552.723,Z 856.271,A -85,B 0,C 180,E1 3141.363,E2 3141.363} C_VEL
LIN {X 0,Y 552.517,Z 865.989,A -85,B 0,C 180,E1 3145.299,E2 3145.299} C_VEL
LIN {X 0,Y 552.49,Z 869.512,A -85,B 0,C 180,E1 3148.434,E2 3148.434} C_VEL
LIN {X 0,Y 552.621,Z 869.513,A -85,B 0,C 180,E1 3151.563,E2 3151.563} C_VEL
LIN {X 0,Y 552.538,Z 865.994,A -85,B 0,C 180,E1 3154.698,E2 3154.698} C_VEL
LIN {X 0,Y 552.676,Z 856.278,A -85,B 0,C 180,E1 3158.635,E2 3158.635} C_VEL
LIN {X 0,Y 552.821,Z 841.988,A -85,B 0,C 180,E1 3162.211,E2 3162.211} C_VEL
LIN {X 0,Y 553.388,Z 823.158,A -85,B 0,C 180,E1 3165.546,E2 3165.546} C_VEL
LIN {X 0,Y 554.231,Z 797.99,A -85,B 0,C 180,E1 3168.841,E2 3168.841} C_VEL
LIN {X 0,Y 555.369,Z 768.144,A -85,B 0,C 180,E1 3171.726,E2 3171.726} C_VEL
LIN {X 0,Y 556.559,Z 736.29,A -85,B 0,C 180,E1 3173.995,E2 3173.995} C_VEL
LIN {X 0,Y 557.662,Z 701.892,A -85,B 0,C 180,E1 3175.736,E2 3175.736} C_VEL
LIN {X 0,Y 558.577,Z 665.634,A -85,B 0,C 180,E1 3176.905,E2 3176.905} C_VEL
LIN {X 0,Y 557.993,Z 595.546,A -85,B 0,C 180,E1 3178.051,E2 3178.051} C_VEL
LIN {X 0,Y 552.147,Z 580.66,A -85,B 0,C 180,E1 3178.696,E2 3178.696} C_VEL
LIN {X 0,Y 551.949,Z 580.66,A -85,B 0,C 180,E1 3185.035,E2 3185.035} C_VEL
LIN {X 0,Y 551.869,Z 580.66,A -85,B 0,C 180,E1 3191.009,E2 3191.009} C_VEL
LIN {X 0,Y 551.973,Z 580.66,A -85,B 0,C 180,E1 3196.887,E2 3196.887} C_VEL
LIN {X 0,Y 551.962,Z 580.66,A -85,B 0,C 180,E1 3203.026,E2 3203.026} C_VEL
LIN {X 0,Y 551.92,Z 580.66,A -85,B 0,C 180,E1 3208.703,E2 3208.703} C_VEL
LIN {X 0,Y 552.082,Z 580.66,A -85,B 0,C 180,E1 3214.411,E2 3214.411} C_VEL
LIN {X 0,Y 552.199,Z 580.66,A -85,B 0,C 180,E1 3220.856,E2 3220.856} C_VEL
LIN {X 0,Y 551.926,Z 580.66,A -85,B 0,C 180,E1 3225.754,E2 3225.754} C_VEL
LIN {X 0,Y 552.149,Z 580.66,A -85,B 0,C 180,E1 3230.56,E2 3230.56} C_VEL
LIN {X 0,Y 552.277,Z 580.66,A -85,B 0,C 180,E1 3235.296,E2 3235.296} C_VEL
LIN {X 0,Y 552.295,Z 580.66,A -85,B 0,C 180,E1 3239.997,E2 3239.997} C_VEL
LIN {X 0,Y 552.337,Z 580.66,A -85,B 0,C 180,E1 3244.698,E2 3244.698} C_VEL
LIN {X 0,Y 552.128,Z 580.66,A -85,B 0,C 180,E1 3250.319,E2 3250.319} C_VEL
LIN {X 0,Y 552.071,Z 580.66,A -85,B 0,C 180,E1 3255.858,E2 3255.858} C_VEL
LIN {X 0,Y 552.05,Z 580.66,A -85,B 0,C 180,E1 3261.675,E2 3261.675} C_VEL
LIN {X 0,Y 551.948,Z 580.66,A -85,B 0,C 180,E1 3267.689,E2 3267.689} C_VEL
LIN {X 0,Y 552.01,Z 580.66,A -85,B 0,C 180,E1 3273.136,E2 3273.136} C_VEL
LIN {X 0,Y 551.799,Z 580.66,A -85,B 0,C 180,E1 3278.967,E2 3278.967} C_VEL
LIN {X 0,Y 551.895,Z 580.66,A -85,B 0,C 180,E1 3284.697,E2 3284.697} C_VEL
LIN {X 0,Y 551.925,Z 580.66,A -85,B 0,C 180,E1 3289.944,E2 3289.944} C_VEL
LIN {X 0,Y 551.945,Z 580.66,A -85,B 0,C 180,E1 3295.091,E2 3295.091} C_VEL
LIN {X 0,Y 551.966,Z 580.66,A -85,B 0,C 180,E1 3301.01,E2 3301.01} C_VEL
LIN {X 0,Y 552.008,Z 580.66,A -85,B 0,C 180,E1 3305.795,E2 3305.795} C_VEL
LIN {X 0,Y 552.198,Z 581.158,A -85,B 0,C 180,E1 3308.635,E2 3308.635} C_VEL
LIN {X 0,Y 555.698,Z 598.894,A -85,B 0,C 180,E1 3309.697,E2 3309.697} C_VEL
LIN {X 0,Y 554.662,Z 631.279,A -85,B 0,C 180,E1 3311.784,E2 3311.784} C_VEL
LIN {X 0,Y 553.828,Z 658.849,A -85,B 0,C 180,E1 3314.311,E2 3314.311} C_VEL
LIN {X 0,Y 553.111,Z 681.43,A -85,B 0,C 180,E1 3317.195,E2 3317.195} C_VEL
LIN {X 0,Y 552.777,Z 698.461,A -85,B 0,C 180,E1 3320.234,E2 3320.234} C_VEL
LIN {X 0,Y 552.575,Z 710.217,A -85,B 0,C 180,E1 3323.337,E2 3323.337} C_VEL
LIN {X 0,Y 552.548,Z 717.9,A -85,B 0,C 180,E1 3326.87,E2 3326.87} C_VEL
LIN {X 0,Y 552.481,Z 719.995,A -85,B 0,C 180,E1 3330.001,E2 3330.001} C_VEL
LIN {X 0,Y 552.564,Z 717.761,A -85,B 0,C 180,E1 3333.132,E2 3333.132} C_VEL
LIN {X 0,Y 552.635,Z 709.948,A -85,B 0,C 180,E1 3336.665,E2 3336.665} C_VEL
LIN {X 0,Y 552.842,Z 696.339,A -85,B 0,C 180,E1 3340.11,E2 3340.11} C_VEL
LIN {X 0,Y 553.26,Z 678.13,A -85,B 0,C 180,E1 3343.205,E2 3343.205} C_VEL
LIN {X 0,Y 553.913,Z 654.926,A -85,B 0,C 180,E1 3346.012,E2 3346.012} C_VEL
LIN {X 0,Y 554.781,Z 627.453,A -85,B 0,C 180,E1 3348.409,E2 3348.409} C_VEL
LIN {X 0,Y 555.516,Z 593.506,A -85,B 0,C 180,E1 3350.506,E2 3350.506} C_VEL
LIN {X 0,Y 552.224,Z 580.66,A -85,B 0,C 180,E1 3351.371,E2 3351.371} C_VEL
LIN {X 0,Y 552.006,Z 580.66,A -85,B 0,C 180,E1 3355.937,E2 3355.937} C_VEL
LIN {X 0,Y 551.86,Z 580.66,A -85,B 0,C 180,E1 3362.056,E2 3362.056} C_VEL
LIN {X 0,Y 552.032,Z 580.66,A -85,B 0,C 180,E1 3367.571,E2 3367.571} C_VEL
LIN {X 0,Y 551.851,Z 580.66,A -85,B 0,C 180,E1 3373.125,E2 3373.125} C_VEL
LIN {X 0,Y 551.967,Z 580.66,A -85,B 0,C 180,E1 3379.003,E2 3379.003} C_VEL
LIN {X 0,Y 551.923,Z 580.66,A -85,B 0,C 180,E1 3385.105,E2 3385.105} C_VEL
LIN {X 0,Y 551.913,Z 580.66,A -85,B 0,C 180,E1 3391.032,E2 3391.032} C_VEL
LIN {X 0,Y 551.977,Z 580.66,A -85,B 0,C 180,E1 3395.796,E2 3395.796} C_VEL
LIN {X 0,Y 552.219,Z 580.66,A -85,B 0,C 180,E1 3400.863,E2 3400.863} C_VEL
LIN {X 0,Y 551.878,Z 580.66,A -85,B 0,C 180,E1 3405.758,E2 3405.758} C_VEL
LIN {X 0,Y 552.126,Z 580.66,A -85,B 0,C 180,E1 3410.566,E2 3410.566} C_VEL
LIN {X 0,Y 552.298,Z 580.66,A -85,B 0,C 180,E1 3415.302,E2 3415.302} C_VEL
LIN {X 0,Y 552.319,Z 580.66,A -85,B 0,C 180,E1 3420.003,E2 3420.003} C_VEL
LIN {X 0,Y 552.295,Z 580.66,A -85,B 0,C 180,E1 3424.704,E2 3424.704} C_VEL
LIN {X 0,Y 552.142,Z 580.66,A -85,B 0,C 180,E1 3430.313,E2 3430.313} C_VEL
LIN {X 0,Y 552.056,Z 580.66,A -85,B 0,C 180,E1 3435.865,E2 3435.865} C_VEL
LIN {X 0,Y 552.069,Z 580.66,A -85,B 0,C 180,E1 3439.666,E2 3439.666} C_VEL
LIN {X 0,Y 548.053,Z 580.66,A -85,B 0,C 180,E1 3441.435,E2 3441.435} C_VEL
LIN {X 0,Y 544.079,Z 580.66,A -85,B 0,C 180,E1 3443.229,E2 3443.229} C_VEL
LIN {X 0,Y 544.077,Z 580.66,A -85,B 0,C 180,E1 3448.132,E2 3448.132} C_VEL
LIN {X 0,Y 544.067,Z 580.66,A -85,B 0,C 180,E1 3453.691,E2 3453.691} C_VEL
LIN {X 0,Y 543.914,Z 580.66,A -85,B 0,C 180,E1 3459.65,E2 3459.65} C_VEL
LIN {X 0,Y 544.009,Z 580.66,A -85,B 0,C 180,E1 3466.153,E2 3466.153} C_VEL
LIN {X 0,Y 544.092,Z 580.66,A -85,B 0,C 180,E1 3472.4,E2 3472.4} C_VEL
LIN {X 0,Y 544.047,Z 580.66,A -85,B 0,C 180,E1 3478.198,E2 3478.198} C_VEL
LIN {X 0,Y 544.192,Z 580.66,A -85,B 0,C 180,E1 3480.923,E2 3480.923} C_VEL
LIN {X 0,Y 551.863,Z 600.766,A -85,B 0,C 180,E1 3481.685,E2 3481.685} C_VEL
LIN {X 0,Y 551.456,Z 667.46,A -85,B 0,C 180,E1 3482.767,E2 3482.767} C_VEL
LIN {X 0,Y 550.409,Z 703.709,A -85,B 0,C 180,E1 3483.982,E2 3483.982} C_VEL
LIN {X 0,Y 549.168,Z 737.935,A -85,B 0,C 180,E1 3485.767,E2 3485.767} C_VEL
LIN {X 0,Y 547.802,Z 770.606,A -85,B 0,C 180,E1 3488.168,E2 3488.168} C_VEL
LIN {X 0,Y 546.555,Z 799.54,A -85,B 0,C 180,E1 3491.07,E2 3491.07} C_VEL
LIN {X 0,Y 545.656,Z 823.988,A -85,B 0,C 180,E1 3494.357,E2 3494.357} C_VEL
LIN {X 0,Y 545.004,Z 843.902,A -85,B 0,C 180,E1 3498.014,E2 3498.014} C_VEL
LIN {X 0,Y 544.824,Z 857.536,A -85,B 0,C 180,E1 3501.638,E2 3501.638} C_VEL
LIN {X 0,Y 544.643,Z 865.989,A -85,B 0,C 180,E1 3505.231,E2 3505.231} C_VEL
LIN {X 0,Y 544.589,Z 869.512,A -85,B 0,C 180,E1 3508.411,E2 3508.411} C_VEL
LIN {X 0,Y 544.718,Z 869.514,A -85,B 0,C 180,E1 3511.586,E2 3511.586} C_VEL
LIN {X 0,Y 544.597,Z 864.494,A -85,B 0,C 180,E1 3515.564,E2 3515.564} C_VEL
LIN {X 0,Y 544.749,Z 854.945,A -85,B 0,C 180,E1 3519.163,E2 3519.163} C_VEL
LIN {X 0,Y 545.056,Z 840.039,A -85,B 0,C 180,E1 3522.794,E2 3522.794} C_VEL
LIN {X 0,Y 545.706,Z 820.058,A -85,B 0,C 180,E1 3526.25,E2 3526.25} C_VEL
LIN {X 0,Y 546.718,Z 794.838,A -85,B 0,C 180,E1 3529.464,E2 3529.464} C_VEL
LIN {X 0,Y 547.987,Z 765.63,A -85,B 0,C 180,E1 3532.246,E2 3532.246} C_VEL
LIN {X 0,Y 549.426,Z 731.998,A -85,B 0,C 180,E1 3534.597,E2 3534.597} C_VEL
LIN {X 0,Y 550.69,Z 697.313,A -85,B 0,C 180,E1 3536.278,E2 3536.278} C_VEL
LIN {X 0,Y 551.605,Z 661.864,A -85,B 0,C 180,E1 3537.358,E2 3537.358} C_VEL
LIN {X 0,Y 551.082,Z 597.791,A -85,B 0,C 180,E1 3538.402,E2 3538.402} C_VEL
LIN {X 0,Y 544.164,Z 580.66,A -85,B 0,C 180,E1 3539.079,E2 3539.079} C_VEL
LIN {X 0,Y 544.072,Z 580.66,A -85,B 0,C 180,E1 3543.692,E2 3543.692} C_VEL
LIN {X 0,Y 543.911,Z 580.66,A -85,B 0,C 180,E1 3549.646,E2 3549.646} C_VEL
LIN {X 0,Y 544.004,Z 580.66,A -85,B 0,C 180,E1 3556.149,E2 3556.149} C_VEL
LIN {X 0,Y 544.081,Z 580.66,A -85,B 0,C 180,E1 3562.399,E2 3562.399} C_VEL
LIN {X 0,Y 544.024,Z 580.66,A -85,B 0,C 180,E1 3568.196,E2 3568.196} C_VEL
LIN {X 0,Y 544.073,Z 580.66,A -85,B 0,C 180,E1 3573.655,E2 3573.655} C_VEL
LIN {X 0,Y 544.177,Z 580.66,A -85,B 0,C 180,E1 3578.869,E2 3578.869} C_VEL
LIN {X 0,Y 544.213,Z 580.66,A -85,B 0,C 180,E1 3583.9,E2 3583.9} C_VEL
LIN {X 0,Y 544.266,Z 580.66,A -85,B 0,C 180,E1 3590.422,E2 3590.422} C_VEL
LIN {X 0,Y 544.39,Z 580.66,A -85,B 0,C 180,E1 3595.227,E2 3595.227} C_VEL
LIN {X 0,Y 544.394,Z 580.66,A -85,B 0,C 180,E1 3599.997,E2 3599.997} C_VEL
LIN {X 0,Y 544.447,Z 580.66,A -85,B 0,C 180,E1 3604.766,E2 3604.766} C_VEL
LIN {X 0,Y 544.328,Z 580.66,A -85,B 0,C 180,E1 3609.571,E2 3609.571} C_VEL
LIN {X 0,Y 544.288,Z 580.66,A -85,B 0,C 180,E1 3614.445,E2 3614.445} C_VEL
LIN {X 0,Y 544.207,Z 580.66,A -85,B 0,C 180,E1 3619.492,E2 3619.492} C_VEL
LIN {X 0,Y 544.056,Z 580.66,A -85,B 0,C 180,E1 3624.579,E2 3624.579} C_VEL
LIN {X 0,Y 543.979,Z 580.66,A -85,B 0,C 180,E1 3630.698,E2 3630.698} C_VEL
LIN {X 0,Y 543.916,Z 580.66,A -85,B 0,C 180,E1 3635.627,E2 3635.627} C_VEL
LIN {X 0,Y 543.908,Z 580.66,A -85,B 0,C 180,E1 3641.739,E2 3641.739} C_VEL
LIN {X 0,Y 544.069,Z 580.66,A -85,B 0,C 180,E1 3648.272,E2 3648.272} C_VEL
LIN {X 0,Y 543.975,Z 580.66,A -85,B 0,C 180,E1 3654.374,E2 3654.374} C_VEL
LIN {X 0,Y 543.965,Z 580.66,A -85,B 0,C 180,E1 3660.047,E2 3660.047} C_VEL
LIN {X 0,Y 544.094,Z 580.66,A -85,B 0,C 180,E1 3665.42,E2 3665.42} C_VEL
LIN {X 0,Y 544.203,Z 580.66,A -85,B 0,C 180,E1 3668.143,E2 3668.143} C_VEL
LIN {X 0,Y 548.611,Z 599.677,A -85,B 0,C 180,E1 3669.341,E2 3669.341} C_VEL
LIN {X 0,Y 547.357,Z 629.567,A -85,B 0,C 180,E1 3671.31,E2 3671.31} C_VEL
LIN {X 0,Y 546.107,Z 657.706,A -85,B 0,C 180,E1 3673.962,E2 3673.962} C_VEL
LIN {X 0,Y 545.381,Z 680.102,A -85,B 0,C 180,E1 3676.807,E2 3676.807} C_VEL
LIN {X 0,Y 544.974,Z 697.222,A -85,B 0,C 180,E1 3679.835,E2 3679.835} C_VEL
LIN {X 0,Y 544.712,Z 710.215,A -85,B 0,C 180,E1 3683.24,E2 3683.24} C_VEL
LIN {X 0,Y 544.652,Z 717.9,A -85,B 0,C 180,E1 3686.825,E2 3686.825} C_VEL
LIN {X 0,Y 544.582,Z 719.995,A -85,B 0,C 180,E1 3690.001,E2 3690.001} C_VEL
LIN {X 0,Y 544.666,Z 717.763,A -85,B 0,C 180,E1 3693.178,E2 3693.178} C_VEL
LIN {X 0,Y 544.761,Z 709.95,A -85,B 0,C 180,E1 3696.762,E2 3696.762} C_VEL
LIN {X 0,Y 544.981,Z 696.764,A -85,B 0,C 180,E1 3700.169,E2 3700.169} C_VEL
LIN {X 0,Y 545.477,Z 678.134,A -85,B 0,C 180,E1 3703.397,E2 3703.397} C_VEL
LIN {X 0,Y 546.226,Z 654.934,A -85,B 0,C 180,E1 3706.244,E2 3706.244} C_VEL
LIN {X 0,Y 547.46,Z 627.064,A -85,B 0,C 180,E1 3708.793,E2 3708.793} C_VEL
LIN {X 0,Y 548.378,Z 595.473,A -85,B 0,C 180,E1 3710.805,E2 3710.805} C_VEL
LIN {X 0,Y 544.269,Z 580.66,A -85,B 0,C 180,E1 3711.755,E2 3711.755} C_VEL
LIN {X 0,Y 543.951,Z 580.66,A -85,B 0,C 180,E1 3718.138,E2 3718.138} C_VEL
LIN {X 0,Y 543.977,Z 580.66,A -85,B 0,C 180,E1 3723.697,E2 3723.697} C_VEL
LIN {X 0,Y 544.041,Z 580.66,A -85,B 0,C 180,E1 3729.638,E2 3729.638} C_VEL
LIN {X 0,Y 543.973,Z 580.66,A -85,B 0,C 180,E1 3736.156,E2 3736.156} C_VEL
LIN {X 0,Y 544.061,Z 580.66,A -85,B 0,C 180,E1 3742.405,E2 3742.405} C_VEL
LIN {X 0,Y 543.989,Z 580.66,A -85,B 0,C 180,E1 3748.2,E2 3748.2} C_VEL
LIN {X 0,Y 544.042,Z 580.66,A -85,B 0,C 180,E1 3753.66,E2 3753.66} C_VEL
LIN {X 0,Y 544.189,Z 580.66,A -85,B 0,C 180,E1 3758.875,E2 3758.875} C_VEL
LIN {X 0,Y 544.182,Z 580.66,A -85,B 0,C 180,E1 3763.906,E2 3763.906} C_VEL
LIN {X 0,Y 544.238,Z 580.66,A -85,B 0,C 180,E1 3770.428,E2 3770.428} C_VEL
LIN {X 0,Y 544.411,Z 580.66,A -85,B 0,C 180,E1 3775.234,E2 3775.234} C_VEL
LIN {X 0,Y 544.418,Z 580.66,A -85,B 0,C 180,E1 3780.003,E2 3780.003} C_VEL
LIN {X 0,Y 544.401,Z 580.66,A -85,B 0,C 180,E1 3784.773,E2 3784.773} C_VEL
LIN {X 0,Y 544.341,Z 580.66,A -85,B 0,C 180,E1 3789.577,E2 3789.577} C_VEL
LIN {X 0,Y 544.324,Z 580.66,A -85,B 0,C 180,E1 3794.45,E2 3794.45} C_VEL
LIN {X 0,Y 544.168,Z 580.66,A -85,B 0,C 180,E1 3799.655,E2 3799.655} C_VEL
LIN {X 0,Y 544.079,Z 580.66,A -85,B 0,C 180,E1 3803.229,E2 3803.229} C_VEL
LIN {X 0,Y 540.139,Z 580.66,A -85,B 0,C 180,E1 3805.032,E2 3805.032} C_VEL
LIN {X 0,Y 536.101,Z 580.66,A -85,B 0,C 180,E1 3806.86,E2 3806.86} C_VEL
LIN {X 0,Y 536.094,Z 580.66,A -85,B 0,C 180,E1 3812.39,E2 3812.39} C_VEL
LIN {X 0,Y 536.004,Z 580.66,A -85,B 0,C 180,E1 3818.269,E2 3818.269} C_VEL
LIN {X 0,Y 535.969,Z 580.66,A -85,B 0,C 180,E1 3824.737,E2 3824.737} C_VEL
LIN {X 0,Y 536.082,Z 580.66,A -85,B 0,C 180,E1 3829.654,E2 3829.654} C_VEL
LIN {X 0,Y 536.053,Z 580.66,A -85,B 0,C 180,E1 3834.719,E2 3834.719} C_VEL
LIN {X 0,Y 536.262,Z 581.174,A -85,B 0,C 180,E1 3840.488,E2 3840.488} C_VEL
LIN {X 0,Y 544.971,Z 603.787,A -85,B 0,C 180,E1 3841.338,E2 3841.338} C_VEL
LIN {X 0,Y 544.476,Z 666.669,A -85,B 0,C 180,E1 3842.366,E2 3842.366} C_VEL
LIN {X 0,Y 543.269,Z 703.707,A -85,B 0,C 180,E1 3843.614,E2 3843.614} C_VEL
LIN {X 0,Y 541.838,Z 737.932,A -85,B 0,C 180,E1 3845.417,E2 3845.417} C_VEL
LIN {X 0,Y 540.304,Z 770.759,A -85,B 0,C 180,E1 3847.863,E2 3847.863} C_VEL
LIN {X 0,Y 538.916,Z 799.54,A -85,B 0,C 180,E1 3850.791,E2 3850.791} C_VEL
LIN {X 0,Y 537.893,Z 823.984,A -85,B 0,C 180,E1 3854.125,E2 3854.125} C_VEL
LIN {X 0,Y 537.186,Z 843.903,A -85,B 0,C 180,E1 3857.837,E2 3857.837} C_VEL
LIN {X 0,Y 536.938,Z 857.536,A -85,B 0,C 180,E1 3861.514,E2 3861.514} C_VEL
LIN {X 0,Y 536.745,Z 865.988,A -85,B 0,C 180,E1 3865.161,E2 3865.161} C_VEL
LIN {X 0,Y 536.697,Z 869.512,A -85,B 0,C 180,E1 3868.388,E2 3868.388} C_VEL
LIN {X 0,Y 536.844,Z 869.514,A -85,B 0,C 180,E1 3871.609,E2 3871.609} C_VEL
LIN {X 0,Y 536.709,Z 864.494,A -85,B 0,C 180,E1 3875.646,E2 3875.646} C_VEL
LIN {X 0,Y 536.878,Z 854.945,A -85,B 0,C 180,E1 3879.299,E2 3879.299} C_VEL
LIN {X 0,Y 537.234,Z 840.04,A -85,B 0,C 180,E1 3882.983,E2 3882.983} C_VEL
LIN {X 0,Y 538.019,Z 819.128,A -85,B 0,C 180,E1 3886.63,E2 3886.63} C_VEL
LIN {X 0,Y 539.138,Z 794.097,A -85,B 0,C 180,E1 3889.831,E2 3889.831} C_VEL
LIN {X 0,Y 540.624,Z 764.641,A -85,B 0,C 180,E1 3892.651,E2 3892.651} C_VEL
LIN {X 0,Y 542.171,Z 730.83,A -85,B 0,C 180,E1 3895.018,E2 3895.018} C_VEL
LIN {X 0,Y 543.628,Z 695.586,A -85,B 0,C 180,E1 3896.714,E2 3896.714} C_VEL
LIN {X 0,Y 544.595,Z 662.043,A -85,B 0,C 180,E1 3897.736,E2 3897.736} C_VEL
LIN {X 0,Y 543.989,Z 599.826,A -85,B 0,C 180,E1 3898.777,E2 3898.777} C_VEL
LIN {X 0,Y 536.227,Z 580.66,A -85,B 0,C 180,E1 3899.555,E2 3899.555} C_VEL
LIN {X 0,Y 536.022,Z 580.66,A -85,B 0,C 180,E1 3905.276,E2 3905.276} C_VEL
LIN {X 0,Y 535.955,Z 580.66,A -85,B 0,C 180,E1 3910.52,E2 3910.52} C_VEL
LIN {X 0,Y 536.042,Z 580.66,A -85,B 0,C 180,E1 3917.042,E2 3917.042} C_VEL
LIN {X 0,Y 536.151,Z 580.66,A -85,B 0,C 180,E1 3921.998,E2 3921.998} C_VEL
LIN {X 0,Y 536.076,Z 580.66,A -85,B 0,C 180,E1 3927.667,E2 3927.667} C_VEL
LIN {X 0,Y 536.149,Z 580.66,A -85,B 0,C 180,E1 3933.235,E2 3933.235} C_VEL
LIN {X 0,Y 536.214,Z 580.66,A -85,B 0,C 180,E1 3938.539,E2 3938.539} C_VEL
LIN {X 0,Y 536.3,Z 580.66,A -85,B 0,C 180,E1 3943.656,E2 3943.656} C_VEL
LIN {X 0,Y 536.347,Z 580.66,A -85,B 0,C 180,E1 3950.279,E2 3950.279} C_VEL
LIN {X 0,Y 536.486,Z 580.66,A -85,B 0,C 180,E1 3955.157,E2 3955.157} C_VEL
LIN {X 0,Y 536.501,Z 580.66,A -85,B 0,C 180,E1 3959.997,E2 3959.997} C_VEL
LIN {X 0,Y 536.531,Z 580.66,A -85,B 0,C 180,E1 3964.837,E2 3964.837} C_VEL
LIN {X 0,Y 536.349,Z 580.66,A -85,B 0,C 180,E1 3970.057,E2 3970.057} C_VEL
LIN {X 0,Y 536.349,Z 580.66,A -85,B 0,C 180,E1 3974.663,E2 3974.663} C_VEL
LIN {X 0,Y 536.296,Z 580.66,A -85,B 0,C 180,E1 3979.729,E2 3979.729} C_VEL
LIN {X 0,Y 536.06,Z 580.66,A -85,B 0,C 180,E1 3985.747,E2 3985.747} C_VEL
LIN {X 0,Y 536.07,Z 580.66,A -85,B 0,C 180,E1 3990.437,E2 3990.437} C_VEL
LIN {X 0,Y 535.99,Z 580.66,A -85,B 0,C 180,E1 3996.236,E2 3996.236} C_VEL
LIN {X 0,Y 535.937,Z 580.66,A -85,B 0,C 180,E1 4002.504,E2 4002.504} C_VEL
LIN {X 0,Y 536.059,Z 580.66,A -85,B 0,C 180,E1 4007.504,E2 4007.504} C_VEL
LIN {X 0,Y 536.09,Z 580.66,A -85,B 0,C 180,E1 4013.768,E2 4013.768} C_VEL
LIN {X 0,Y 536.055,Z 580.66,A -85,B 0,C 180,E1 4019.559,E2 4019.559} C_VEL
LIN {X 0,Y 536.148,Z 580.66,A -85,B 0,C 180,E1 4025.031,E2 4025.031} C_VEL
LIN {X 0,Y 536.27,Z 581.226,A -85,B 0,C 180,E1 4027.706,E2 4027.706} C_VEL
LIN {X 0,Y 541.573,Z 599.896,A -85,B 0,C 180,E1 4028.943,E2 4028.943} C_VEL
LIN {X 0,Y 540.171,Z 630.129,A -85,B 0,C 180,E1 4030.947,E2 4030.947} C_VEL
LIN {X 0,Y 538.742,Z 657.243,A -85,B 0,C 180,E1 4033.527,E2 4033.527} C_VEL
LIN {X 0,Y 537.618,Z 680.204,A -85,B 0,C 180,E1 4036.613,E2 4036.613} C_VEL
LIN {X 0,Y 537.111,Z 698.068,A -85,B 0,C 180,E1 4039.864,E2 4039.864} C_VEL
LIN {X 0,Y 536.828,Z 710.213,A -85,B 0,C 180,E1 4043.14,E2 4043.14} C_VEL
LIN {X 0,Y 536.759,Z 717.9,A -85,B 0,C 180,E1 4046.778,E2 4046.778} C_VEL
LIN {X 0,Y 536.705,Z 719.995,A -85,B 0,C 180,E1 4050.001,E2 4050.001} C_VEL
LIN {X 0,Y 536.771,Z 717.765,A -85,B 0,C 180,E1 4053.224,E2 4053.224} C_VEL
LIN {X 0,Y 536.871,Z 709.952,A -85,B 0,C 180,E1 4056.862,E2 4056.862} C_VEL
LIN {X 0,Y 537.156,Z 696.444,A -85,B 0,C 180,E1 4060.387,E2 4060.387} C_VEL
LIN {X 0,Y 537.859,Z 675.599,A -85,B 0,C 180,E1 4064.004,E2 4064.004} C_VEL
LIN {X 0,Y 538.983,Z 652.662,A -85,B 0,C 180,E1 4066.887,E2 4066.887} C_VEL
LIN {X 0,Y 540.421,Z 624.995,A -85,B 0,C 180,E1 4069.365,E2 4069.365} C_VEL
LIN {X 0,Y 541.126,Z 597.129,A -85,B 0,C 180,E1 4071.141,E2 4071.141} C_VEL
LIN {X 0,Y 536.295,Z 580.66,A -85,B 0,C 180,E1 4072.296,E2 4072.296} C_VEL
LIN {X 0,Y 535.996,Z 580.66,A -85,B 0,C 180,E1 4078.594,E2 4078.594} C_VEL
LIN {X 0,Y 536.022,Z 580.66,A -85,B 0,C 180,E1 4084.266,E2 4084.266} C_VEL
LIN {X 0,Y 536.177,Z 580.66,A -85,B 0,C 180,E1 4088.254,E2 4088.254} C_VEL
LIN {X 0,Y 535.943,Z 580.66,A -85,B 0,C 180,E1 4094.739,E2 4094.739} C_VEL
LIN {X 0,Y 536.048,Z 580.66,A -85,B 0,C 180,E1 4099.658,E2 4099.658} C_VEL
LIN {X 0,Y 536.02,Z 580.66,A -85,B 0,C 180,E1 4104.724,E2 4104.724} C_VEL
LIN {X 0,Y 535.996,Z 580.66,A -85,B 0,C 180,E1 4110.777,E2 4110.777} C_VEL
LIN {X 0,Y 536.162,Z 580.66,A -85,B 0,C 180,E1 4116.801,E2 4116.801} C_VEL
LIN {X 0,Y 536.372,Z 580.66,A -85,B 0,C 180,E1 4121.978,E2 4121.978} C_VEL
LIN {X 0,Y 536.28,Z 580.66,A -85,B 0,C 180,E1 4128.644,E2 4128.644} C_VEL
LIN {X 0,Y 536.507,Z 580.66,A -85,B 0,C 180,E1 4135.163,E2 4135.163} C_VEL
LIN {X 0,Y 536.524,Z 580.66,A -85,B 0,C 180,E1 4140.003,E2 4140.003} C_VEL
LIN {X 0,Y 536.487,Z 580.66,A -85,B 0,C 180,E1 4144.843,E2 4144.843} C_VEL
LIN {X 0,Y 536.395,Z 580.66,A -85,B 0,C 180,E1 4150.069,E2 4150.069} C_VEL
LIN {X 0,Y 536.377,Z 580.66,A -85,B 0,C 180,E1 4154.669,E2 4154.669} C_VEL
LIN {X 0,Y 536.283,Z 580.66,A -85,B 0,C 180,E1 4159.736,E2 4159.736} C_VEL
LIN {X 0,Y 536.079,Z 580.66,A -85,B 0,C 180,E1 4165.745,E2 4165.745} C_VEL
LIN {X 0,Y 536.101,Z 580.66,A -85,B 0,C 180,E1 4166.86,E2 4166.86} C_VEL
LIN {X 0,Y 532.018,Z 580.66,A -85,B 0,C 180,E1 4168.689,E2 4168.689} C_VEL
LIN {X 0,Y 528.113,Z 580.66,A -85,B 0,C 180,E1 4170.546,E2 4170.546} C_VEL
LIN {X 0,Y 528.12,Z 580.66,A -85,B 0,C 180,E1 4174.852,E2 4174.852} C_VEL
LIN {X 0,Y 527.992,Z 580.66,A -85,B 0,C 180,E1 4181.097,E2 4181.097} C_VEL
LIN {X 0,Y 528.089,Z 580.66,A -85,B 0,C 180,E1 4186.703,E2 4186.703} C_VEL
LIN {X 0,Y 528.188,Z 580.66,A -85,B 0,C 180,E1 4193.123,E2 4193.123} C_VEL
LIN {X 0,Y 528.193,Z 580.66,A -85,B 0,C 180,E1 4199.053,E2 4199.053} C_VEL
LIN {X 0,Y 528.323,Z 580.66,A -85,B 0,C 180,E1 4200.046,E2 4200.046} C_VEL
LIN {X 0,Y 538.071,Z 606.212,A -85,B 0,C 180,E1 4200.972,E2 4200.972} C_VEL
LIN {X 0,Y 537.433,Z 667.533,A -85,B 0,C 180,E1 4201.997,E2 4201.997} C_VEL
LIN {X 0,Y 536.094,Z 704.727,A -85,B 0,C 180,E1 4203.28,E2 4203.28} C_VEL
LIN {X 0,Y 534.506,Z 739.627,A -85,B 0,C 180,E1 4205.169,E2 4205.169} C_VEL
LIN {X 0,Y 532.736,Z 772.823,A -85,B 0,C 180,E1 4207.724,E2 4207.724} C_VEL
LIN {X 0,Y 531.226,Z 801.286,A -85,B 0,C 180,E1 4210.718,E2 4210.718} C_VEL
LIN {X 0,Y 530.077,Z 825.304,A -85,B 0,C 180,E1 4214.097,E2 4214.097} C_VEL
LIN {X 0,Y 529.387,Z 843.903,A -85,B 0,C 180,E1 4217.655,E2 4217.655} C_VEL
LIN {X 0,Y 529.078,Z 857.536,A -85,B 0,C 180,E1 4221.387,E2 4221.387} C_VEL
LIN {X 0,Y 528.861,Z 865.987,A -85,B 0,C 180,E1 4225.088,E2 4225.088} C_VEL
LIN {X 0,Y 528.795,Z 869.512,A -85,B 0,C 180,E1 4228.363,E2 4228.363} C_VEL
LIN {X 0,Y 528.941,Z 869.514,A -85,B 0,C 180,E1 4231.633,E2 4231.633} C_VEL
LIN {X 0,Y 528.834,Z 864.494,A -85,B 0,C 180,E1 4235.73,E2 4235.73} C_VEL
LIN {X 0,Y 528.997,Z 854.944,A -85,B 0,C 180,E1 4239.439,E2 4239.439} C_VEL
LIN {X 0,Y 529.444,Z 840.041,A -85,B 0,C 180,E1 4243.178,E2 4243.178} C_VEL
LIN {X 0,Y 530.294,Z 819.387,A -85,B 0,C 180,E1 4246.841,E2 4246.841} C_VEL
LIN {X 0,Y 531.554,Z 793.898,A -85,B 0,C 180,E1 4250.149,E2 4250.149} C_VEL
LIN {X 0,Y 533.194,Z 764.388,A -85,B 0,C 180,E1 4253.006,E2 4253.006} C_VEL
LIN {X 0,Y 534.976,Z 730.367,A -85,B 0,C 180,E1 4255.406,E2 4255.406} C_VEL
LIN {X 0,Y 536.52,Z 696.086,A -85,B 0,C 180,E1 4257.077,E2 4257.077} C_VEL
LIN {X 0,Y 537.634,Z 660.706,A -85,B 0,C 180,E1 4258.158,E2 4258.158} C_VEL
LIN {X 0,Y 537.176,Z 602.285,A -85,B 0,C 180,E1 4259.14,E2 4259.14} C_VEL
LIN {X 0,Y 528.28,Z 580.66,A -85,B 0,C 180,E1 4260.002,E2 4260.002} C_VEL
LIN {X 0,Y 528.134,Z 580.66,A -85,B 0,C 180,E1 4264.847,E2 4264.847} C_VEL
LIN {X 0,Y 527.991,Z 580.66,A -85,B 0,C 180,E1 4271.093,E2 4271.093} C_VEL
LIN {X 0,Y 528.091,Z 580.66,A -85,B 0,C 180,E1 4276.703,E2 4276.703} C_VEL
LIN {X 0,Y 528.148,Z 580.66,A -85,B 0,C 180,E1 4281.055,E2 4281.055} C_VEL
LIN {X 0,Y 528.128,Z 580.66,A -85,B 0,C 180,E1 4287.12,E2 4287.12} C_VEL
LIN {X 0,Y 528.186,Z 580.66,A -85,B 0,C 180,E1 4292.798,E2 4292.798} C_VEL
LIN {X 0,Y 528.31,Z 580.66,A -85,B 0,C 180,E1 4298.202,E2 4298.202} C_VEL
LIN {X 0,Y 528.414,Z 580.66,A -85,B 0,C 180,E1 4303.405,E2 4303.405} C_VEL
LIN {X 0,Y 528.454,Z 580.66,A -85,B 0,C 180,E1 4310.133,E2 4310.133} C_VEL
LIN {X 0,Y 528.592,Z 580.66,A -85,B 0,C 180,E1 4315.084,E2 4315.084} C_VEL
LIN {X 0,Y 528.601,Z 580.66,A -85,B 0,C 180,E1 4319.997,E2 4319.997} C_VEL
LIN {X 0,Y 528.621,Z 580.66,A -85,B 0,C 180,E1 4324.909,E2 4324.909} C_VEL
LIN {X 0,Y 528.484,Z 580.66,A -85,B 0,C 180,E1 4329.861,E2 4329.861} C_VEL
LIN {X 0,Y 528.435,Z 580.66,A -85,B 0,C 180,E1 4334.888,E2 4334.888} C_VEL
LIN {X 0,Y 528.356,Z 580.66,A -85,B 0,C 180,E1 4340.038,E2 4340.038} C_VEL
LIN {X 0,Y 528.181,Z 580.66,A -85,B 0,C 180,E1 4345.369,E2 4345.369} C_VEL
LIN {X 0,Y 528.136,Z 580.66,A -85,B 0,C 180,E1 4351.008,E2 4351.008} C_VEL
LIN {X 0,Y 528.048,Z 580.66,A -85,B 0,C 180,E1 4356.87,E2 4356.87} C_VEL
LIN {X 0,Y 528.005,Z 580.66,A -85,B 0,C 180,E1 4363.297,E2 4363.297} C_VEL
LIN {X 0,Y 528.126,Z 580.66,A -85,B 0,C 180,E1 4368.92,E2 4368.92} C_VEL
LIN {X 0,Y 528.099,Z 580.66,A -85,B 0,C 180,E1 4375.15,E2 4375.15} C_VEL
LIN {X 0,Y 528.181,Z 580.66,A -85,B 0,C 180,E1 4380.946,E2 4380.946} C_VEL
LIN {X 0,Y 528.323,Z 580.66,A -85,B 0,C 180,E1 4387.18,E2 4387.18} C_VEL
LIN {X 0,Y 534.474,Z 602.768,A -85,B 0,C 180,E1 4388.679,E2 4388.679} C_VEL
LIN {X 0,Y 532.943,Z 632.097,A -85,B 0,C 180,E1 4390.678,E2 4390.678} C_VEL
LIN {X 0,Y 531.337,Z 659.039,A -85,B 0,C 180,E1 4393.312,E2 4393.312} C_VEL
LIN {X 0,Y 530.068,Z 681.726,A -85,B 0,C 180,E1 4396.429,E2 4396.429} C_VEL
LIN {X 0,Y 529.319,Z 698.554,A -85,B 0,C 180,E1 4399.713,E2 4399.713} C_VEL
LIN {X 0,Y 528.913,Z 711.355,A -85,B 0,C 180,E1 4403.449,E2 4403.449} C_VEL
LIN {X 0,Y 528.864,Z 718.082,A -85,B 0,C 180,E1 4406.865,E2 4406.865} C_VEL
LIN {X 0,Y 528.806,Z 719.995,A -85,B 0,C 180,E1 4410.001,E2 4410.001} C_VEL
LIN {X 0,Y 528.895,Z 717.766,A -85,B 0,C 180,E1 4413.272,E2 4413.272} C_VEL
LIN {X 0,Y 528.996,Z 709.954,A -85,B 0,C 180,E1 4416.964,E2 4416.964} C_VEL
LIN {X 0,Y 529.427,Z 696.178,A -85,B 0,C 180,E1 4420.733,E2 4420.733} C_VEL
LIN {X 0,Y 530.258,Z 678.593,A -85,B 0,C 180,E1 4423.98,E2 4423.98} C_VEL
LIN {X 0,Y 531.51,Z 656.569,A -85,B 0,C 180,E1 4426.883,E2 4426.883} C_VEL
LIN {X 0,Y 533.058,Z 629.649,A -85,B 0,C 180,E1 4429.428,E2 4429.428} C_VEL
LIN {X 0,Y 533.978,Z 599.008,A -85,B 0,C 180,E1 4431.473,E2 4431.473} C_VEL
LIN {X 0,Y 528.34,Z 580.66,A -85,B 0,C 180,E1 4432.776,E2 4432.776} C_VEL
LIN {X 0,Y 528.104,Z 580.66,A -85,B 0,C 180,E1 4439.062,E2 4439.062} C_VEL
LIN {X 0,Y 528.122,Z 580.66,A -85,B 0,C 180,E1 4444.851,E2 4444.851} C_VEL
LIN {X 0,Y 528.061,Z 580.66,A -85,B 0,C 180,E1 4451.09,E2 4451.09} C_VEL
LIN {X 0,Y 528.056,Z 580.66,A -85,B 0,C 180,E1 4456.708,E2 4456.708} C_VEL
LIN {X 0,Y 528.156,Z 580.66,A -85,B 0,C 180,E1 4463.127,E2 4463.127} C_VEL
LIN {X 0,Y 528.095,Z 580.66,A -85,B 0,C 180,E1 4469.053,E2 4469.053} C_VEL
LIN {X 0,Y 528.211,Z 580.66,A -85,B 0,C 180,E1 4474.632,E2 4474.632} C_VEL
LIN {X 0,Y 528.443,Z 580.66,A -85,B 0,C 180,E1 4480.442,E2 4480.442} C_VEL
LIN {X 0,Y 528.145,Z 580.66,A -85,B 0,C 180,E1 4486.266,E2 4486.266} C_VEL
LIN {X 0,Y 528.416,Z 580.66,A -85,B 0,C 180,E1 4491.795,E2 4491.795} C_VEL
LIN {X 0,Y 528.631,Z 580.66,A -85,B 0,C 180,E1 4497.513,E2 4497.513} C_VEL
LIN {X 0,Y 528.664,Z 580.66,A -85,B 0,C 180,E1 4503.275,E2 4503.275} C_VEL
LIN {X 0,Y 528.514,Z 580.66,A -85,B 0,C 180,E1 4509.866,E2 4509.866} C_VEL
LIN {X 0,Y 528.458,Z 580.66,A -85,B 0,C 180,E1 4514.893,E2 4514.893} C_VEL
LIN {X 0,Y 528.354,Z 580.66,A -85,B 0,C 180,E1 4520.044,E2 4520.044} C_VEL
LIN {X 0,Y 528.201,Z 580.66,A -85,B 0,C 180,E1 4525.375,E2 4525.375} C_VEL
LIN {X 0,Y 528.113,Z 580.66,A -85,B 0,C 180,E1 4530.546,E2 4530.546} C_VEL
LIN {X 0,Y 525.635,Z 580.66,A -85,B 0,C 180,E1 4531.948,E2 4531.948} C_VEL
LIN {X 0,Y 520.116,Z 580.66,A -85,B 0,C 180,E1 4534.292,E2 4534.292} C_VEL
LIN {X 0,Y 520.107,Z 580.66,A -85,B 0,C 180,E1 4539.664,E2 4539.664} C_VEL
LIN {X 0,Y 520.17,Z 580.66,A -85,B 0,C 180,E1 4545.876,E2 4545.876} C_VEL
LIN {X 0,Y 520.219,Z 580.66,A -85,B 0,C 180,E1 4551.552,E2 4551.552} C_VEL
LIN {X 0,Y 520.228,Z 580.66,A -85,B 0,C 180,E1 4557.263,E2 4557.263} C_VEL
LIN {X 0,Y 520.348,Z 580.66,A -85,B 0,C 180,E1 4559.63,E2 4559.63} C_VEL
LIN {X 0,Y 531.021,Z 606.9,A -85,B 0,C 180,E1 4560.582,E2 4560.582} C_VEL
LIN {X 0,Y 530.497,Z 666.763,A -85,B 0,C 180,E1 4561.576,E2 4561.576} C_VEL
LIN {X 0,Y 529.063,Z 703.701,A -85,B 0,C 180,E1 4562.848,E2 4562.848} C_VEL
LIN {X 0,Y 527.304,Z 737.925,A -85,B 0,C 180,E1 4564.693,E2 4564.693} C_VEL
LIN {X 0,Y 525.423,Z 771.204,A -85,B 0,C 180,E1 4567.241,E2 4567.241} C_VEL
LIN {X 0,Y 523.697,Z 799.539,A -85,B 0,C 180,E1 4570.21,E2 4570.21} C_VEL
LIN {X 0,Y 522.364,Z 823.982,A -85,B 0,C 180,E1 4573.64,E2 4573.64} C_VEL
LIN {X 0,Y 521.548,Z 843.903,A -85,B 0,C 180,E1 4577.466,E2 4577.466} C_VEL
LIN {X 0,Y 521.197,Z 857.536,A -85,B 0,C 180,E1 4581.256,E2 4581.256} C_VEL
LIN {X 0,Y 520.963,Z 865.987,A -85,B 0,C 180,E1 4585.014,E2 4585.014} C_VEL
LIN {X 0,Y 520.908,Z 869.513,A -85,B 0,C 180,E1 4588.339,E2 4588.339} C_VEL
LIN {X 0,Y 521.047,Z 869.515,A -85,B 0,C 180,E1 4591.658,E2 4591.658} C_VEL
LIN {X 0,Y 520.969,Z 864.493,A -85,B 0,C 180,E1 4595.817,E2 4595.817} C_VEL
LIN {X 0,Y 521.158,Z 854.944,A -85,B 0,C 180,E1 4599.582,E2 4599.582} C_VEL
LIN {X 0,Y 521.631,Z 840.042,A -85,B 0,C 180,E1 4603.379,E2 4603.379} C_VEL
LIN {X 0,Y 522.574,Z 819.85,A -85,B 0,C 180,E1 4607.025,E2 4607.025} C_VEL
LIN {X 0,Y 523.993,Z 793.898,A -85,B 0,C 180,E1 4610.453,E2 4610.453} C_VEL
LIN {X 0,Y 525.819,Z 764.154,A -85,B 0,C 180,E1 4613.369,E2 4613.369} C_VEL
LIN {X 0,Y 527.757,Z 730.368,A -85,B 0,C 180,E1 4615.779,E2 4615.779} C_VEL
LIN {X 0,Y 529.486,Z 695.161,A -85,B 0,C 180,E1 4617.505,E2 4617.505} C_VEL
LIN {X 0,Y 530.679,Z 660.665,A -85,B 0,C 180,E1 4618.562,E2 4618.562} C_VEL
LIN {X 0,Y 530.009,Z 604.112,A -85,B 0,C 180,E1 4619.508,E2 4619.508} C_VEL
LIN {X 0,Y 520.334,Z 580.66,A -85,B 0,C 180,E1 4620.42,E2 4620.42} C_VEL
LIN {X 0,Y 520.137,Z 580.66,A -85,B 0,C 180,E1 4625.678,E2 4625.678} C_VEL
LIN {X 0,Y 520.085,Z 580.66,A -85,B 0,C 180,E1 4631.857,E2 4631.857} C_VEL
LIN {X 0,Y 520.206,Z 580.66,A -85,B 0,C 180,E1 4638.151,E2 4638.151} C_VEL
LIN {X 0,Y 520.19,Z 580.66,A -85,B 0,C 180,E1 4644.309,E2 4644.309} C_VEL
LIN {X 0,Y 520.258,Z 580.66,A -85,B 0,C 180,E1 4650.467,E2 4650.467} C_VEL
LIN {X 0,Y 520.304,Z 580.66,A -85,B 0,C 180,E1 4656.043,E2 4656.043} C_VEL
LIN {X 0,Y 520.521,Z 580.66,A -85,B 0,C 180,E1 4661.403,E2 4661.403} C_VEL
LIN {X 0,Y 520.455,Z 580.66,A -85,B 0,C 180,E1 4668.288,E2 4668.288} C_VEL
LIN {X 0,Y 520.698,Z 580.66,A -85,B 0,C 180,E1 4673.341,E2 4673.341} C_VEL
LIN {X 0,Y 520.867,Z 580.66,A -85,B 0,C 180,E1 4678.337,E2 4678.337} C_VEL
LIN {X 0,Y 520.705,Z 580.66,A -85,B 0,C 180,E1 4684.984,E2 4684.984} C_VEL
LIN {X 0,Y 520.58,Z 580.66,A -85,B 0,C 180,E1 4690.012,E2 4690.012} C_VEL
LIN {X 0,Y 520.503,Z 580.66,A -85,B 0,C 180,E1 4695.12,E2 4695.12} C_VEL
LIN {X 0,Y 520.413,Z 580.66,A -85,B 0,C 180,E1 4700.357,E2 4700.357} C_VEL
LIN {X 0,Y 520.216,Z 580.66,A -85,B 0,C 180,E1 4705.954,E2 4705.954} C_VEL
LIN {X 0,Y 520.214,Z 580.66,A -85,B 0,C 180,E1 4711.468,E2 4711.468} C_VEL
LIN {X 0,Y 520.055,Z 580.66,A -85,B 0,C 180,E1 4717.534,E2 4717.534} C_VEL
LIN {X 0,Y 520.101,Z 580.66,A -85,B 0,C 180,E1 4723.508,E2 4723.508} C_VEL
LIN {X 0,Y 520.223,Z 580.66,A -85,B 0,C 180,E1 4728.943,E2 4728.943} C_VEL
LIN {X 0,Y 520.155,Z 580.66,A -85,B 0,C 180,E1 4734.539,E2 4734.539} C_VEL
LIN {X 0,Y 520.221,Z 580.66,A -85,B 0,C 180,E1 4740.467,E2 4740.467} C_VEL
LIN {X 0,Y 520.384,Z 580.66,A -85,B 0,C 180,E1 4746.668,E2 4746.668} C_VEL
LIN {X 0,Y 527.378,Z 605.154,A -85,B 0,C 180,E1 4748.378,E2 4748.378} C_VEL
LIN {X 0,Y 525.679,Z 635.379,A -85,B 0,C 180,E1 4750.51,E2 4750.51} C_VEL
LIN {X 0,Y 523.988,Z 660.571,A -85,B 0,C 180,E1 4753.05,E2 4753.05} C_VEL
LIN {X 0,Y 522.642,Z 681.653,A -85,B 0,C 180,E1 4755.97,E2 4755.97} C_VEL
LIN {X 0,Y 521.675,Z 699.752,A -85,B 0,C 180,E1 4759.527,E2 4759.527} C_VEL
LIN {X 0,Y 521.109,Z 712.328,A -85,B 0,C 180,E1 4763.35,E2 4763.35} C_VEL
LIN {X 0,Y 520.995,Z 718.449,A -85,B 0,C 180,E1 4766.681,E2 4766.681} C_VEL
LIN {X 0,Y 520.932,Z 720.417,A -85,B 0,C 180,E1 4770.001,E2 4770.001} C_VEL
LIN {X 0,Y 521.039,Z 717.187,A -85,B 0,C 180,E1 4774.153,E2 4774.153} C_VEL
LIN {X 0,Y 521.355,Z 708.592,A -85,B 0,C 180,E1 4777.903,E2 4777.903} C_VEL
LIN {X 0,Y 521.989,Z 693.919,A -85,B 0,C 180,E1 4781.676,E2 4781.676} C_VEL
LIN {X 0,Y 523.137,Z 674.418,A -85,B 0,C 180,E1 4785.047,E2 4785.047} C_VEL
LIN {X 0,Y 524.718,Z 650.089,A -85,B 0,C 180,E1 4788.023,E2 4788.023} C_VEL
LIN {X 0,Y 526.441,Z 622.651,A -85,B 0,C 180,E1 4790.395,E2 4790.395} C_VEL
LIN {X 0,Y 526.705,Z 600.182,A -85,B 0,C 180,E1 4791.867,E2 4791.867} C_VEL
LIN {X 0,Y 520.39,Z 580.66,A -85,B 0,C 180,E1 4793.311,E2 4793.311} C_VEL
LIN {X 0,Y 520.176,Z 580.66,A -85,B 0,C 180,E1 4799.548,E2 4799.548} C_VEL
LIN {X 0,Y 520.2,Z 580.66,A -85,B 0,C 180,E1 4805.699,E2 4805.699} C_VEL
LIN {X 0,Y 520.158,Z 580.66,A -85,B 0,C 180,E1 4811.049,E2 4811.049} C_VEL
LIN {X 0,Y 520.141,Z 580.66,A -85,B 0,C 180,E1 4816.491,E2 4816.491} C_VEL
LIN {X 0,Y 520.197,Z 580.66,A -85,B 0,C 180,E1 4822.478,E2 4822.478} C_VEL
LIN {X 0,Y 520.161,Z 580.66,A -85,B 0,C 180,E1 4828.528,E2 4828.528} C_VEL
LIN {X 0,Y 520.246,Z 580.66,A -85,B 0,C 180,E1 4834.215,E2 4834.215} C_VEL
LIN {X 0,Y 520.447,Z 580.66,A -85,B 0,C 180,E1 4839.644,E2 4839.644} C_VEL
LIN {X 0,Y 520.305,Z 580.66,A -85,B 0,C 180,E1 4844.874,E2 4844.874} C_VEL
LIN {X 0,Y 520.508,Z 580.66,A -85,B 0,C 180,E1 4850.285,E2 4850.285} C_VEL
LIN {X 0,Y 520.705,Z 580.66,A -85,B 0,C 180,E1 4855.016,E2 4855.016} C_VEL
LIN {X 0,Y 520.734,Z 580.66,A -85,B 0,C 180,E1 4860.003,E2 4860.003} C_VEL
LIN {X 0,Y 520.675,Z 580.66,A -85,B 0,C 180,E1 4864.991,E2 4864.991} C_VEL
LIN {X 0,Y 520.612,Z 580.66,A -85,B 0,C 180,E1 4870.017,E2 4870.017} C_VEL
LIN {X 0,Y 520.517,Z 580.66,A -85,B 0,C 180,E1 4875.126,E2 4875.126} C_VEL
LIN {X 0,Y 520.412,Z 580.66,A -85,B 0,C 180,E1 4880.364,E2 4880.364} C_VEL
LIN {X 0,Y 520.24,Z 580.66,A -85,B 0,C 180,E1 4885.953,E2 4885.953} C_VEL
LIN {X 0,Y 520.203,Z 580.66,A -85,B 0,C 180,E1 4891.476,E2 4891.476} C_VEL
LIN {X 0,Y 520.116,Z 580.66,A -85,B 0,C 180,E1 4894.292,E2 4894.292} C_VEL
LIN {X 0,Y 518.807,Z 580.66,A -85,B 0,C 180,E1 4895.245,E2 4895.245} C_VEL
LIN {X 0,Y 512.242,Z 580.66,A -85,B 0,C 180,E1 4897.842,E2 4897.842} C_VEL
LIN {X 0,Y 512.168,Z 580.66,A -85,B 0,C 180,E1 4898.088,E2 4898.088} C_VEL
LIN {X 0,Y 512.158,Z 580.66,A -85,B 0,C 180,E1 4902.661,E2 4902.661} C_VEL
